REGION Network 3: E-Stop / Call: 运行 模式 area 1 - Create 新的 OpMode
   // 介绍：设置和管理操作操作模式OPMode，有几个OPMode就需要调用几次，每次调用都需要对其与HMI的关系进行定义。
   // 一个OPMode至少需要一个HMI/pannei控制；
   // 一个HMI/Panel可以控制多个OPMode；
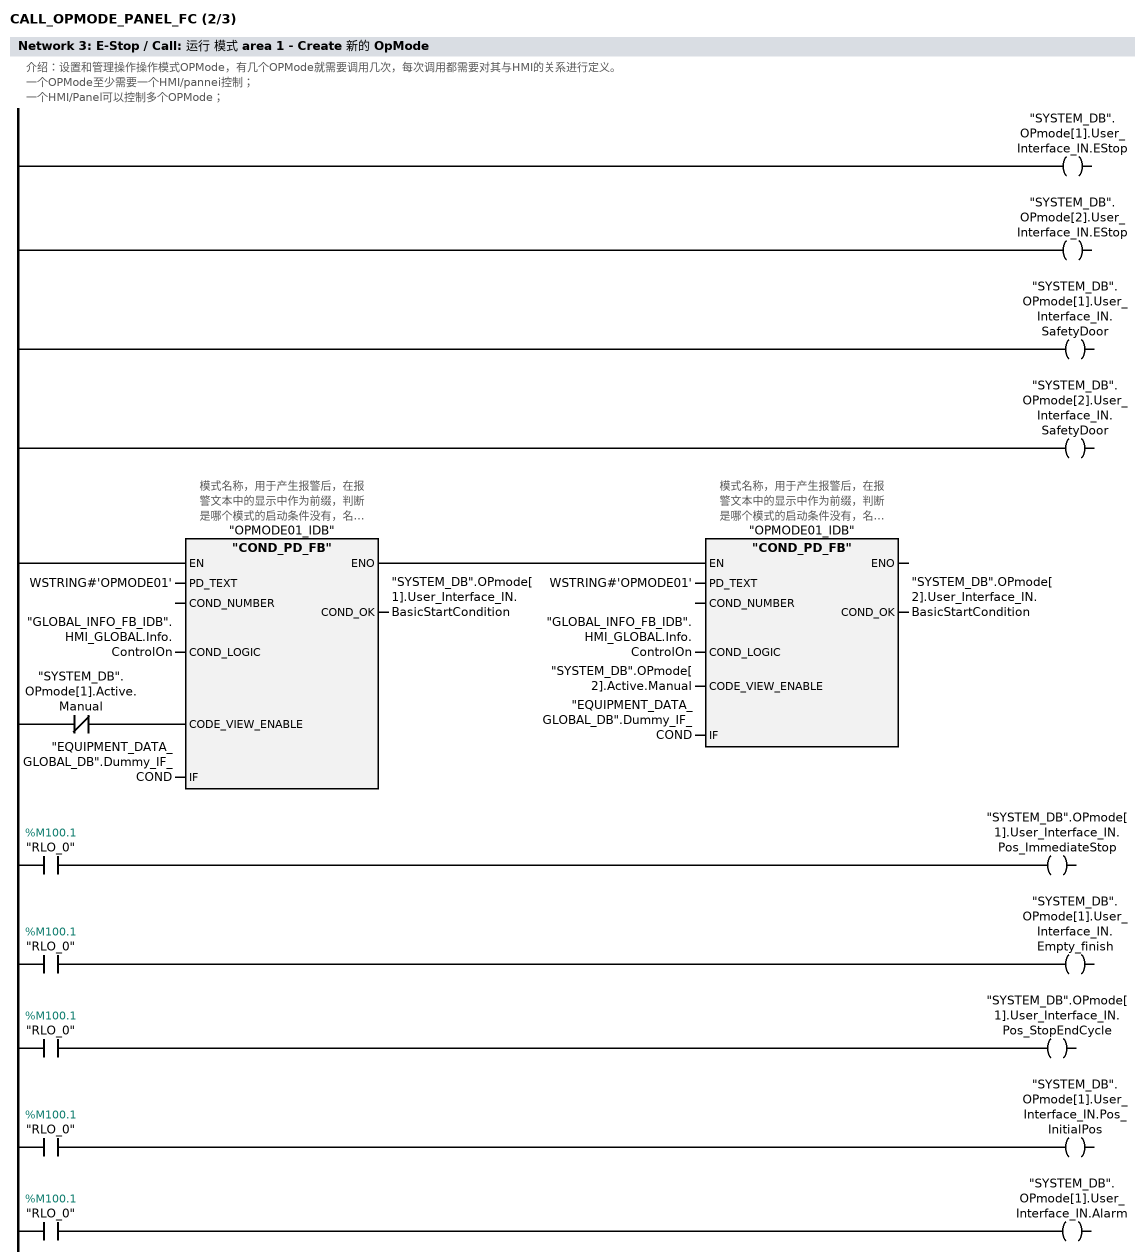
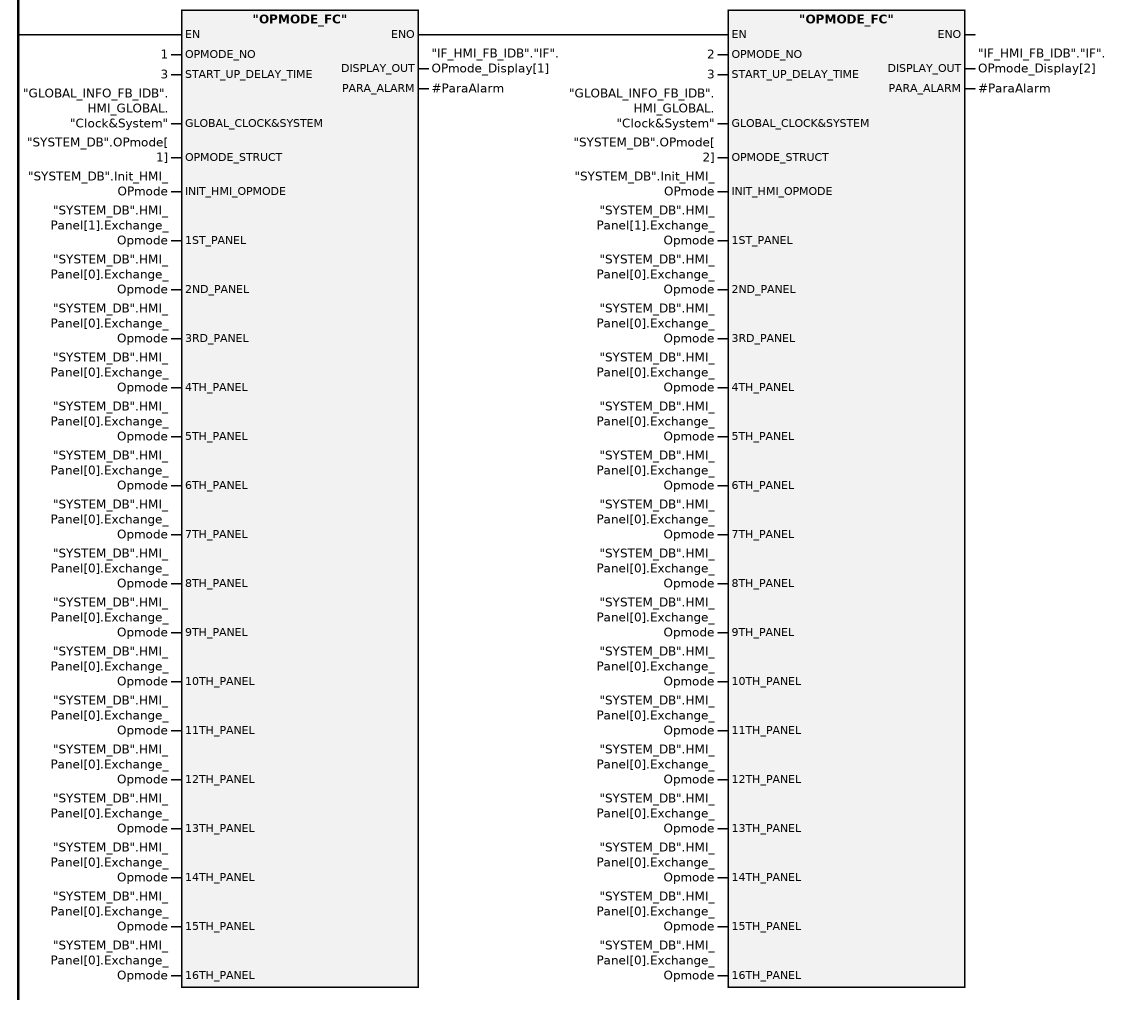
   RUNG wire#powerrail
      Coil( "SYSTEM_DB".OPmode[1].User_Interface_IN.EStop )
   END_RUNG
   RUNG wire#powerrail
      Coil( "SYSTEM_DB".OPmode[2].User_Interface_IN.EStop )
   END_RUNG
   RUNG wire#powerrail
      Coil( "SYSTEM_DB".OPmode[1].User_Interface_IN.SafetyDoor )
   END_RUNG
   RUNG wire#powerrail
      Coil( "SYSTEM_DB".OPmode[2].User_Interface_IN.SafetyDoor )
   END_RUNG
   RUNG wire#powerrail
      "OPMODE01_IDB"(CODE_VIEW_ENABLE := wire#w1, PD_TEXT := WSTRING#'OPMODE01', COND_NUMBER :=, COND_LOGIC := "GLOBAL_INFO_FB_IDB".HMI_GLOBAL.Info.ControlOn, "IF" := "EQUIPMENT_DATA_GLOBAL_DB".Dummy_IF_COND, COND_OK => "SYSTEM_DB".OPmode[1].User_Interface_IN.BasicStartCondition)   // 模式名称，用于产生报警后，在报警文本中的显示中作为前缀，判断是哪个模式的启动条件没有，名称已经预先填写在了对应DB块数据中
      "OPMODE01_IDB"(PD_TEXT := WSTRING#'OPMODE01', COND_NUMBER :=, COND_LOGIC := "GLOBAL_INFO_FB_IDB".HMI_GLOBAL.Info.ControlOn, CODE_VIEW_ENABLE := "SYSTEM_DB".OPmode[2].Active.Manual, "IF" := "EQUIPMENT_DATA_GLOBAL_DB".Dummy_IF_COND, COND_OK => "SYSTEM_DB".OPmode[2].User_Interface_IN.BasicStartCondition)   // 模式名称，用于产生报警后，在报警文本中的显示中作为前缀，判断是哪个模式的启动条件没有，名称已经预先填写在了对应DB块数据中
   END_RUNG
   RUNG wire#powerrail
      I_Contact( "SYSTEM_DB".OPmode[1].Active.Manual )
   END_RUNG wire#w1
   RUNG wire#powerrail
      Contact( "RLO_0" )
      Coil( "SYSTEM_DB".OPmode[1].User_Interface_IN.Pos_ImmediateStop )
   END_RUNG
   RUNG wire#powerrail
      Contact( "RLO_0" )
      Coil( "SYSTEM_DB".OPmode[1].User_Interface_IN.Empty_finish )
   END_RUNG
   RUNG wire#powerrail
      Contact( "RLO_0" )
      Coil( "SYSTEM_DB".OPmode[1].User_Interface_IN.Pos_StopEndCycle )
   END_RUNG
   RUNG wire#powerrail
      Contact( "RLO_0" )
      Coil( "SYSTEM_DB".OPmode[1].User_Interface_IN.Pos_InitialPos )
   END_RUNG
   RUNG wire#powerrail
      Contact( "RLO_0" )
      Coil( "SYSTEM_DB".OPmode[1].User_Interface_IN.Alarm )
   END_RUNG
   RUNG wire#powerrail
      "OPMODE_FC"(OPMODE_NO := 1, START_UP_DELAY_TIME := 3, "GLOBAL_CLOCK&SYSTEM" := "GLOBAL_INFO_FB_IDB".HMI_GLOBAL."Clock&System", OPMODE_STRUCT := "SYSTEM_DB".OPmode[1], INIT_HMI_OPMODE := "SYSTEM_DB".Init_HMI_OPmode, "1ST_PANEL" := "SYSTEM_DB".HMI_Panel[1].Exchange_Opmode, "2ND_PANEL" := "SYSTEM_DB".HMI_Panel[0].Exchange_Opmode, "3RD_PANEL" := "SYSTEM_DB".HMI_Panel[0].Exchange_Opmode, "4TH_PANEL" := "SYSTEM_DB".HMI_Panel[0].Exchange_Opmode, "5TH_PANEL" := "SYSTEM_DB".HMI_Panel[0].Exchange_Opmode, "6TH_PANEL" := "SYSTEM_DB".HMI_Panel[0].Exchange_Opmode, "7TH_PANEL" := "SYSTEM_DB".HMI_Panel[0].Exchange_Opmode, "8TH_PANEL" := "SYSTEM_DB".HMI_Panel[0].Exchange_Opmode, "9TH_PANEL" := "SYSTEM_DB".HMI_Panel[0].Exchange_Opmode, "10TH_PANEL" := "SYSTEM_DB".HMI_Panel[0].Exchange_Opmode, "11TH_PANEL" := "SYSTEM_DB".HMI_Panel[0].Exchange_Opmode, "12TH_PANEL" := "SYSTEM_DB".HMI_Panel[0].Exchange_Opmode, "13TH_PANEL" := "SYSTEM_DB".HMI_Panel[0].Exchange_Opmode, "14TH_PANEL" := "SYSTEM_DB".HMI_Panel[0].Exchange_Opmode, "15TH_PANEL" := "SYSTEM_DB".HMI_Panel[0].Exchange_Opmode, "16TH_PANEL" := "SYSTEM_DB".HMI_Panel[0].Exchange_Opmode, DISPLAY_OUT => "IF_HMI_FB_IDB"."IF".OPmode_Display[1], PARA_ALARM => #ParaAlarm)
      "OPMODE_FC"(OPMODE_NO := 2, START_UP_DELAY_TIME := 3, "GLOBAL_CLOCK&SYSTEM" := "GLOBAL_INFO_FB_IDB".HMI_GLOBAL."Clock&System", OPMODE_STRUCT := "SYSTEM_DB".OPmode[2], INIT_HMI_OPMODE := "SYSTEM_DB".Init_HMI_OPmode, "1ST_PANEL" := "SYSTEM_DB".HMI_Panel[1].Exchange_Opmode, "2ND_PANEL" := "SYSTEM_DB".HMI_Panel[0].Exchange_Opmode, "3RD_PANEL" := "SYSTEM_DB".HMI_Panel[0].Exchange_Opmode, "4TH_PANEL" := "SYSTEM_DB".HMI_Panel[0].Exchange_Opmode, "5TH_PANEL" := "SYSTEM_DB".HMI_Panel[0].Exchange_Opmode, "6TH_PANEL" := "SYSTEM_DB".HMI_Panel[0].Exchange_Opmode, "7TH_PANEL" := "SYSTEM_DB".HMI_Panel[0].Exchange_Opmode, "8TH_PANEL" := "SYSTEM_DB".HMI_Panel[0].Exchange_Opmode, "9TH_PANEL" := "SYSTEM_DB".HMI_Panel[0].Exchange_Opmode, "10TH_PANEL" := "SYSTEM_DB".HMI_Panel[0].Exchange_Opmode, "11TH_PANEL" := "SYSTEM_DB".HMI_Panel[0].Exchange_Opmode, "12TH_PANEL" := "SYSTEM_DB".HMI_Panel[0].Exchange_Opmode, "13TH_PANEL" := "SYSTEM_DB".HMI_Panel[0].Exchange_Opmode, "14TH_PANEL" := "SYSTEM_DB".HMI_Panel[0].Exchange_Opmode, "15TH_PANEL" := "SYSTEM_DB".HMI_Panel[0].Exchange_Opmode, "16TH_PANEL" := "SYSTEM_DB".HMI_Panel[0].Exchange_Opmode, DISPLAY_OUT => "IF_HMI_FB_IDB"."IF".OPmode_Display[2], PARA_ALARM => #ParaAlarm)
   END_RUNG
   // the same network as SCL:
   "SYSTEM_DB".OPmode[1].User_Interface_IN.EStop := TRUE;
   "SYSTEM_DB".OPmode[2].User_Interface_IN.EStop := TRUE;
   "SYSTEM_DB".OPmode[1].User_Interface_IN.SafetyDoor := TRUE;
   "SYSTEM_DB".OPmode[2].User_Interface_IN.SafetyDoor := TRUE;
   "OPMODE01_IDB"(PD_TEXT := WSTRING#'OPMODE01',   // "COND_PD_FB": 模式名称，用于产生报警后，在报警文本中的显示中作为前缀，判断是哪个模式的启动条件没有，名称已经预先填写在了对应DB块数据中
                  COND_LOGIC := "GLOBAL_INFO_FB_IDB".HMI_GLOBAL.Info.ControlOn,
                  CODE_VIEW_ENABLE := NOT "SYSTEM_DB".OPmode[1].Active.Manual,
                  "IF" := "EQUIPMENT_DATA_GLOBAL_DB".Dummy_IF_COND,
                  COND_OK => "SYSTEM_DB".OPmode[1].User_Interface_IN.BasicStartCondition,
                  ENO => #_w1);
   IF #_w1 THEN
       "OPMODE01_IDB"(PD_TEXT := WSTRING#'OPMODE01',   // "COND_PD_FB": 模式名称，用于产生报警后，在报警文本中的显示中作为前缀，判断是哪个模式的启动条件没有，名称已经预先填写在了对应DB块数据中
                      COND_LOGIC := "GLOBAL_INFO_FB_IDB".HMI_GLOBAL.Info.ControlOn,
                      CODE_VIEW_ENABLE := "SYSTEM_DB".OPmode[2].Active.Manual,
                      "IF" := "EQUIPMENT_DATA_GLOBAL_DB".Dummy_IF_COND,
                      COND_OK => "SYSTEM_DB".OPmode[2].User_Interface_IN.BasicStartCondition);
   END_IF;
   "SYSTEM_DB".OPmode[1].User_Interface_IN.Pos_ImmediateStop := "RLO_0";
   "SYSTEM_DB".OPmode[1].User_Interface_IN.Empty_finish := "RLO_0";
   "SYSTEM_DB".OPmode[1].User_Interface_IN.Pos_StopEndCycle := "RLO_0";
   "SYSTEM_DB".OPmode[1].User_Interface_IN.Pos_InitialPos := "RLO_0";
   "SYSTEM_DB".OPmode[1].User_Interface_IN.Alarm := "RLO_0";
   "OPMODE_FC"(OPMODE_NO := 1,
               START_UP_DELAY_TIME := 3,
               "GLOBAL_CLOCK&SYSTEM" := "GLOBAL_INFO_FB_IDB".HMI_GLOBAL."Clock&System",
               OPMODE_STRUCT := "SYSTEM_DB".OPmode[1],
               INIT_HMI_OPMODE := "SYSTEM_DB".Init_HMI_OPmode,
               "1ST_PANEL" := "SYSTEM_DB".HMI_Panel[1].Exchange_Opmode,
               "2ND_PANEL" := "SYSTEM_DB".HMI_Panel[0].Exchange_Opmode,
               "3RD_PANEL" := "SYSTEM_DB".HMI_Panel[0].Exchange_Opmode,
               "4TH_PANEL" := "SYSTEM_DB".HMI_Panel[0].Exchange_Opmode,
               "5TH_PANEL" := "SYSTEM_DB".HMI_Panel[0].Exchange_Opmode,
               "6TH_PANEL" := "SYSTEM_DB".HMI_Panel[0].Exchange_Opmode,
               "7TH_PANEL" := "SYSTEM_DB".HMI_Panel[0].Exchange_Opmode,
               "8TH_PANEL" := "SYSTEM_DB".HMI_Panel[0].Exchange_Opmode,
               "9TH_PANEL" := "SYSTEM_DB".HMI_Panel[0].Exchange_Opmode,
               "10TH_PANEL" := "SYSTEM_DB".HMI_Panel[0].Exchange_Opmode,
               "11TH_PANEL" := "SYSTEM_DB".HMI_Panel[0].Exchange_Opmode,
               "12TH_PANEL" := "SYSTEM_DB".HMI_Panel[0].Exchange_Opmode,
               "13TH_PANEL" := "SYSTEM_DB".HMI_Panel[0].Exchange_Opmode,
               "14TH_PANEL" := "SYSTEM_DB".HMI_Panel[0].Exchange_Opmode,
               "15TH_PANEL" := "SYSTEM_DB".HMI_Panel[0].Exchange_Opmode,
               "16TH_PANEL" := "SYSTEM_DB".HMI_Panel[0].Exchange_Opmode,
               DISPLAY_OUT => "IF_HMI_FB_IDB"."IF".OPmode_Display[1],
               PARA_ALARM => #ParaAlarm,
               ENO => #_w2);
   IF #_w2 THEN
       "OPMODE_FC"(OPMODE_NO := 2,
                   START_UP_DELAY_TIME := 3,
                   "GLOBAL_CLOCK&SYSTEM" := "GLOBAL_INFO_FB_IDB".HMI_GLOBAL."Clock&System",
                   OPMODE_STRUCT := "SYSTEM_DB".OPmode[2],
                   INIT_HMI_OPMODE := "SYSTEM_DB".Init_HMI_OPmode,
                   "1ST_PANEL" := "SYSTEM_DB".HMI_Panel[1].Exchange_Opmode,
                   "2ND_PANEL" := "SYSTEM_DB".HMI_Panel[0].Exchange_Opmode,
                   "3RD_PANEL" := "SYSTEM_DB".HMI_Panel[0].Exchange_Opmode,
                   "4TH_PANEL" := "SYSTEM_DB".HMI_Panel[0].Exchange_Opmode,
                   "5TH_PANEL" := "SYSTEM_DB".HMI_Panel[0].Exchange_Opmode,
                   "6TH_PANEL" := "SYSTEM_DB".HMI_Panel[0].Exchange_Opmode,
                   "7TH_PANEL" := "SYSTEM_DB".HMI_Panel[0].Exchange_Opmode,
                   "8TH_PANEL" := "SYSTEM_DB".HMI_Panel[0].Exchange_Opmode,
                   "9TH_PANEL" := "SYSTEM_DB".HMI_Panel[0].Exchange_Opmode,
                   "10TH_PANEL" := "SYSTEM_DB".HMI_Panel[0].Exchange_Opmode,
                   "11TH_PANEL" := "SYSTEM_DB".HMI_Panel[0].Exchange_Opmode,
                   "12TH_PANEL" := "SYSTEM_DB".HMI_Panel[0].Exchange_Opmode,
                   "13TH_PANEL" := "SYSTEM_DB".HMI_Panel[0].Exchange_Opmode,
                   "14TH_PANEL" := "SYSTEM_DB".HMI_Panel[0].Exchange_Opmode,
                   "15TH_PANEL" := "SYSTEM_DB".HMI_Panel[0].Exchange_Opmode,
                   "16TH_PANEL" := "SYSTEM_DB".HMI_Panel[0].Exchange_Opmode,
                   DISPLAY_OUT => "IF_HMI_FB_IDB"."IF".OPmode_Display[2],
                   PARA_ALARM => #ParaAlarm);
   END_IF;
END_REGION

REGION Network 4: Aufruf: HMI Schnittstelle / Call HMI_IF_FB
   // 介绍：HMI与PLC系统的接口功能块，
   // 此块用来管理所有的HMIheOPMode操作模式的接口，用户不需要对此做任何修改。
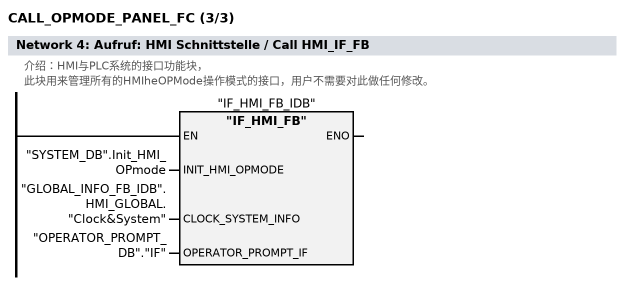
   RUNG wire#powerrail
      "IF_HMI_FB_IDB"(INIT_HMI_OPMODE := "SYSTEM_DB".Init_HMI_OPmode, CLOCK_SYSTEM_INFO := "GLOBAL_INFO_FB_IDB".HMI_GLOBAL."Clock&System", OPERATOR_PROMPT_IF := "OPERATOR_PROMPT_DB"."IF")
   END_RUNG
   // the same network as SCL:
   "IF_HMI_FB_IDB"(INIT_HMI_OPMODE := "SYSTEM_DB".Init_HMI_OPmode,   // "IF_HMI_FB"
                   CLOCK_SYSTEM_INFO := "GLOBAL_INFO_FB_IDB".HMI_GLOBAL."Clock&System",
                   OPERATOR_PROMPT_IF := "OPERATOR_PROMPT_DB"."IF");
END_REGION
END_FUNCTION

FUNCTION "IO映射" : Void   // FC4, LAD
{ S7_Optimized_Access := 'TRUE' }
// stored: SetENOAutomatically false
   VAR_TEMP
      LOOP : Int;
      Value : Byte;
      LOOP_1 : Int;
      Value_1 : Byte;
   END_VAR
BEGIN

REGION Network 1 (SCL)
   // 输入映射
   FOR #LOOP := 0 TO 10 BY 1 DO
       #Value := PEEK(area := 16#81, dbNumber := 0, byteOffset := #LOOP);
       POKE(area := 16#84,
            dbNumber := 12,
            byteOffset := #LOOP,
            value := #Value);
   END_FOR;
END_REGION

REGION Network 2 (SCL)
   // 输出映射
   FOR #LOOP_1 := 0 TO 8 BY 1 DO
       #Value_1 := PEEK(area := 16#84, dbNumber := 13, byteOffset := #LOOP_1);
       POKE(area := 16#82,
            dbNumber := 0,
            byteOffset := #LOOP_1,
            value := #Value_1);
   END_FOR;
END_REGION

REGION Network 3
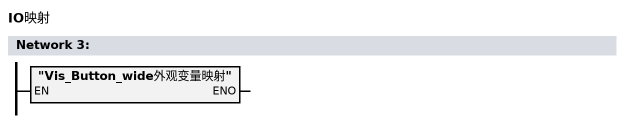
   RUNG wire#powerrail
      "Vis_Button_wide外观变量映射"()
   END_RUNG
   // the same network as SCL:
   "Vis_Button_wide外观变量映射"();
END_REGION
END_FUNCTION

FUNCTION "Vis_Button_wide外观变量映射" : Void   // FC5, LAD
{ S7_Optimized_Access := 'TRUE' }
// stored: SetENOAutomatically false
   VAR_TEMP
      x1 : Bool;
   END_VAR
BEGIN

REGION Network 1
   // 轴1轴2点动速度映射
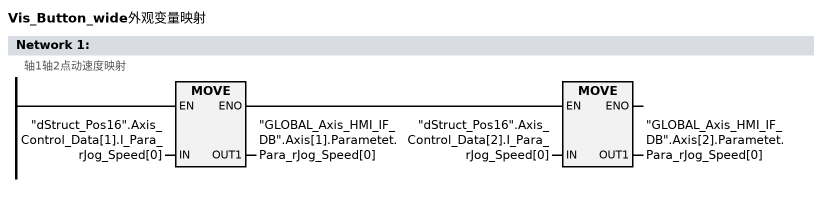
   RUNG wire#powerrail
      Move(in := "dStruct_Pos16".Axis_Control_Data[1].I_Para_rJog_Speed[0], out1 => "GLOBAL_Axis_HMI_IF_DB".Axis[1].Parametet.Para_rJog_Speed[0])
      Move(in := "dStruct_Pos16".Axis_Control_Data[2].I_Para_rJog_Speed[0], out1 => "GLOBAL_Axis_HMI_IF_DB".Axis[2].Parametet.Para_rJog_Speed[0])
   END_RUNG
   // the same network as SCL:
   "GLOBAL_Axis_HMI_IF_DB".Axis[1].Parametet.Para_rJog_Speed[0] := "dStruct_Pos16".Axis_Control_Data[1].I_Para_rJog_Speed[0];
   "GLOBAL_Axis_HMI_IF_DB".Axis[2].Parametet.Para_rJog_Speed[0] := "dStruct_Pos16".Axis_Control_Data[2].I_Para_rJog_Speed[0];
END_REGION

REGION Network 2 (SCL)
   "HMI变量汇总".Vis_Button_wideX1 := "IF_HMI_FB_IDB".IF.HMI[1].Vis_Button_wide.%X1;
   "HMI变量汇总".Vis_Button_wideX2 := "IF_HMI_FB_IDB".IF.HMI[1].Vis_Button_wide.%X2;
   "HMI变量汇总".Vis_Button_wideX3 := "IF_HMI_FB_IDB".IF.HMI[1].Vis_Button_wide.%X3;
   "HMI变量汇总".Vis_Button_wideX4 := "IF_HMI_FB_IDB".IF.HMI[1].Vis_Button_wide.%X4;
   "HMI变量汇总".Vis_Button_wideX5 := "IF_HMI_FB_IDB".IF.HMI[1].Vis_Button_wide.%X5;
   "HMI变量汇总".Vis_Button_wideX6 := "IF_HMI_FB_IDB".IF.HMI[1].Vis_Button_wide.%X6;
   "HMI变量汇总".Vis_Button_wideX7 := "IF_HMI_FB_IDB".IF.HMI[1].Vis_Button_wide.%X7;
   "HMI变量汇总".Vis_Button_wideX8 := "IF_HMI_FB_IDB".IF.HMI[1].Vis_Button_wide.%X8;
   "HMI变量汇总".Vis_Button_wideX9 := "IF_HMI_FB_IDB".IF.HMI[1].Vis_Button_wide.%X9;
   "HMI变量汇总".Vis_Button_wideX10 := "IF_HMI_FB_IDB".IF.HMI[1].Vis_Button_wide.%X10;
   "HMI变量汇总".Vis_Button_wideX11 := "IF_HMI_FB_IDB".IF.HMI[1].Vis_Button_wide.%X11;
   "HMI变量汇总".Vis_Button_wideX12 := "IF_HMI_FB_IDB".IF.HMI[1].Vis_Button_wide.%X12;

   "HMI变量汇总".Vis_Button_small1 := "IF_HMI_FB_IDB".IF.HMI[1].Vis_Button_small.%X1;
   "HMI变量汇总".Vis_Button_small2 := "IF_HMI_FB_IDB".IF.HMI[1].Vis_Button_small.%X2;
   "HMI变量汇总".Vis_Button_small3 := "IF_HMI_FB_IDB".IF.HMI[1].Vis_Button_small.%X3;
   "HMI变量汇总".Vis_Button_small4 := "IF_HMI_FB_IDB".IF.HMI[1].Vis_Button_small.%X4;
   "HMI变量汇总".Vis_Button_small5 := "IF_HMI_FB_IDB".IF.HMI[1].Vis_Button_small.%X5;
   "HMI变量汇总".Vis_Button_small6 := "IF_HMI_FB_IDB".IF.HMI[1].Vis_Button_small.%X6;
   "HMI变量汇总".Vis_Button_small7 := "IF_HMI_FB_IDB".IF.HMI[1].Vis_Button_small.%X7;
   "HMI变量汇总".Vis_Button_small8 := "IF_HMI_FB_IDB".IF.HMI[1].Vis_Button_small.%X8;
   "HMI变量汇总".Vis_Button_small9 := "IF_HMI_FB_IDB".IF.HMI[1].Vis_Button_small.%X9;
   "HMI变量汇总".Vis_Button_small10 := "IF_HMI_FB_IDB".IF.HMI[1].Vis_Button_small.%X10;
   "HMI变量汇总".Vis_Button_small11 := "IF_HMI_FB_IDB".IF.HMI[1].Vis_Button_small.%X11;
   "HMI变量汇总".Vis_Button_small12 := "IF_HMI_FB_IDB".IF.HMI[1].Vis_Button_small.%X12;




   #x1 := "IF_HMI_FB_IDB".IF.StateHeader_ForHMIAnimation[1].%X0;
   #x1 := "IF_HMI_FB_IDB".IF.StateHeader_ForHMIAnimation[1].%X1;
   #x1 := "IF_HMI_FB_IDB".IF.StateHeader_ForHMIAnimation[1].%X2;
   #x1 := "IF_HMI_FB_IDB".IF.StateHeader_ForHMIAnimation[1].%X3;
   #x1 := "IF_HMI_FB_IDB".IF.StateHeader_ForHMIAnimation[1].%X4;
   #x1 := "IF_HMI_FB_IDB".IF.StateHeader_ForHMIAnimation[1].%X5;
   #x1 := "IF_HMI_FB_IDB".IF.StateHeader_ForHMIAnimation[1].%X6;
   #x1 := "IF_HMI_FB_IDB".IF.StateHeader_ForHMIAnimation[1].%X7;
   #x1 := "IF_HMI_FB_IDB".IF.StateHeader_ForHMIAnimation[1].%X8;
   #x1 := "IF_HMI_FB_IDB".IF.StateHeader_ForHMIAnimation[1].%X9;
   #x1 := "IF_HMI_FB_IDB".IF.StateHeader_ForHMIAnimation[1].%X10;
   #x1 := "IF_HMI_FB_IDB".IF.StateHeader_ForHMIAnimation[1].%X11;
   #x1 := "IF_HMI_FB_IDB".IF.StateHeader_ForHMIAnimation[1].%X12;
   #x1 := "IF_HMI_FB_IDB".IF.StateHeader_ForHMIAnimation[1].%X13;
   #x1 := "IF_HMI_FB_IDB".IF.StateHeader_ForHMIAnimation[1].%X14;
   #x1 := "IF_HMI_FB_IDB".IF.StateHeader_ForHMIAnimation[1].%X15;
END_REGION
END_FUNCTION

FUNCTION "OPmode_01" : Void   // FC2, LAD
{ S7_Optimized_Access := 'TRUE' }
// stored: SetENOAutomatically false
BEGIN

REGION Network 1
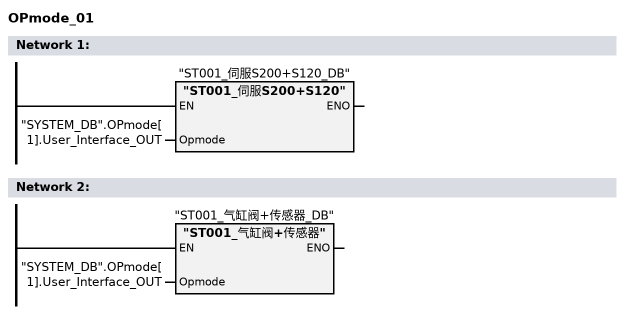
   RUNG wire#powerrail
      "ST001_伺服S200+S120_DB"(Opmode := "SYSTEM_DB".OPmode[1].User_Interface_OUT)
   END_RUNG
   // the same network as SCL:
   "ST001_伺服S200+S120_DB"(Opmode := "SYSTEM_DB".OPmode[1].User_Interface_OUT);   // "ST001_伺服S200+S120"
END_REGION

REGION Network 2
   RUNG wire#powerrail
      "ST001_气缸阀+传感器_DB"(Opmode := "SYSTEM_DB".OPmode[1].User_Interface_OUT)
   END_RUNG
   // the same network as SCL:
   "ST001_气缸阀+传感器_DB"(Opmode := "SYSTEM_DB".OPmode[1].User_Interface_OUT);   // "ST001_气缸阀+传感器"
END_REGION
END_FUNCTION

ORGANIZATION_BLOCK "CyclicInterrupt"   // OB30, LAD, CyclicInterrupt
{ S7_Optimized_Access := 'TRUE' }
// stored: SetENOAutomatically false
   VAR_INPUT
      Initial_Call : Bool;   // Initial call of this OB
      Event_Count : Int;   // Events discarded
   END_VAR
BEGIN

REGION Network 2
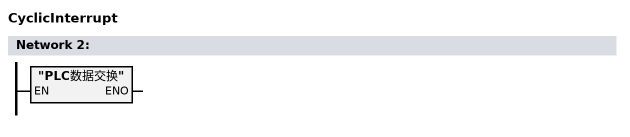
   RUNG wire#powerrail
      "PLC数据交换"()
   END_RUNG
   // the same network as SCL:
   "PLC数据交换"();
END_REGION
END_ORGANIZATION_BLOCK

FUNCTION "PLC数据交换" : Void   // FC1, LAD
{ S7_Optimized_Access := 'TRUE' }
// stored: SetENOAutomatically false
BEGIN

REGION Network 1
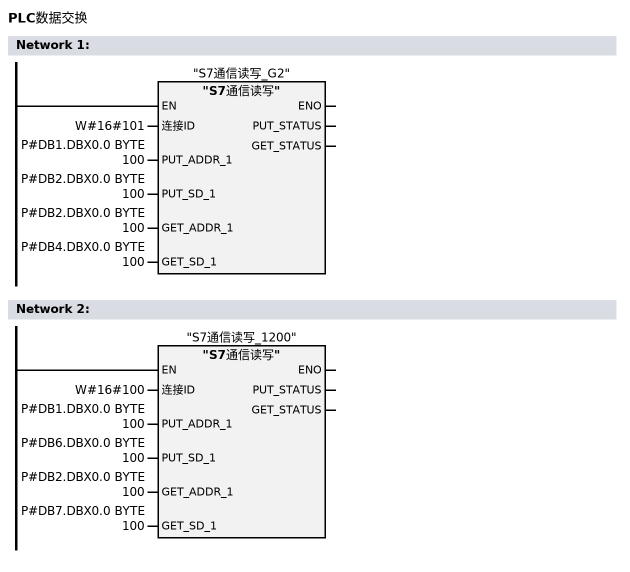
   RUNG wire#powerrail
      "S7通信读写_G2"(连接ID := W#16#101, PUT_ADDR_1 := P#DB1.DBX0.0 BYTE 100, PUT_SD_1 := P#DB2.DBX0.0 BYTE 100, GET_ADDR_1 := P#DB2.DBX0.0 BYTE 100, GET_SD_1 := P#DB4.DBX0.0 BYTE 100, PUT_STATUS =>, GET_STATUS =>)
   END_RUNG
   // the same network as SCL:
   "S7通信读写_G2"(连接ID := W#16#101,   // "S7通信读写"
               PUT_ADDR_1 := P#DB1.DBX0.0 BYTE 100,
               PUT_SD_1 := P#DB2.DBX0.0 BYTE 100,
               GET_ADDR_1 := P#DB2.DBX0.0 BYTE 100,
               GET_SD_1 := P#DB4.DBX0.0 BYTE 100);
END_REGION

REGION Network 2
   RUNG wire#powerrail
      "S7通信读写_1200"(连接ID := W#16#100, PUT_ADDR_1 := P#DB1.DBX0.0 BYTE 100, PUT_SD_1 := P#DB6.DBX0.0 BYTE 100, GET_ADDR_1 := P#DB2.DBX0.0 BYTE 100, GET_SD_1 := P#DB7.DBX0.0 BYTE 100, PUT_STATUS =>, GET_STATUS =>)
   END_RUNG
   // the same network as SCL:
   "S7通信读写_1200"(连接ID := W#16#100,   // "S7通信读写"
                 PUT_ADDR_1 := P#DB1.DBX0.0 BYTE 100,
                 PUT_SD_1 := P#DB6.DBX0.0 BYTE 100,
                 GET_ADDR_1 := P#DB2.DBX0.0 BYTE 100,
                 GET_SD_1 := P#DB7.DBX0.0 BYTE 100);
END_REGION
END_FUNCTION

FUNCTION_BLOCK "S7通信读写"   // FB1, LAD
{ S7_Optimized_Access := 'TRUE' }
// stored: MemoryReserve 100, SetENOAutomatically false
   VAR_INPUT
      连接ID : Word;
   END_VAR
   VAR_OUTPUT
      PUT_STATUS : Word;
      GET_STATUS : Word;
   END_VAR
   VAR_IN_OUT
      PUT_ADDR_1 : Remote;
      PUT_SD_1 : Variant;
      GET_ADDR_1 : Remote;
      GET_SD_1 : Variant;
   END_VAR
   VAR
      PUT_Instance { S7_SetPoint := 'True'} : PUT;
      GET_Instance { S7_SetPoint := 'True'} : GET;
      PUTdone : Bool;
      PUTerror : Bool;
      GETdone : Bool;
      GETerror : Bool;
   END_VAR
BEGIN

REGION Network 1
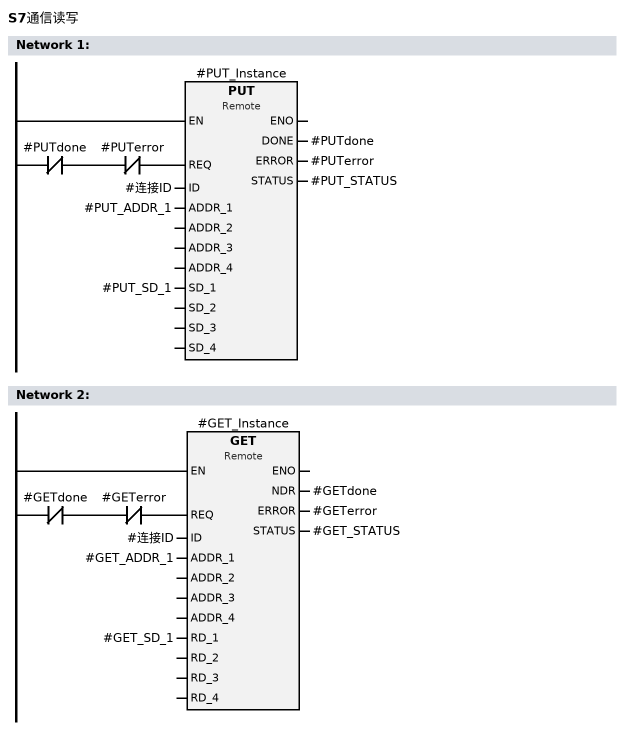
   RUNG wire#powerrail
      { S7_Templates := "[remote_type := Remote, local_type := Variant]" } #PUT_Instance.PUT(REQ := wire#w1, ID := #连接ID, ADDR_1 := #PUT_ADDR_1, ADDR_2 :=, ADDR_3 :=, ADDR_4 :=, SD_1 := #PUT_SD_1, SD_2 :=, SD_3 :=, SD_4 :=, DONE => #PUTdone, ERROR => #PUTerror, STATUS => #PUT_STATUS)
   END_RUNG
   RUNG wire#powerrail
      I_Contact( #PUTdone )
      I_Contact( #PUTerror )
   END_RUNG wire#w1
   // the same network as SCL:
   #PUT_Instance(REQ := NOT #PUTdone AND NOT #PUTerror,   // PUT
                 ID := #连接ID,
                 ADDR_1 := #PUT_ADDR_1,
                 SD_1 := #PUT_SD_1,
                 DONE => #PUTdone,
                 ERROR => #PUTerror,
                 STATUS => #PUT_STATUS);
END_REGION

REGION Network 2
   RUNG wire#powerrail
      { S7_Templates := "[remote_type := Remote, local_type := Variant]" } #GET_Instance.GET(REQ := wire#w1, ID := #连接ID, ADDR_1 := #GET_ADDR_1, ADDR_2 :=, ADDR_3 :=, ADDR_4 :=, RD_1 := #GET_SD_1, RD_2 :=, RD_3 :=, RD_4 :=, NDR => #GETdone, ERROR => #GETerror, STATUS => #GET_STATUS)
   END_RUNG
   RUNG wire#powerrail
      I_Contact( #GETdone )
      I_Contact( #GETerror )
   END_RUNG wire#w1
   // the same network as SCL:
   #GET_Instance(REQ := NOT #GETdone AND NOT #GETerror,   // GET
                 ID := #连接ID,
                 ADDR_1 := #GET_ADDR_1,
                 RD_1 := #GET_SD_1,
                 NDR => #GETdone,
                 ERROR => #GETerror,
                 STATUS => #GET_STATUS);
END_REGION
END_FUNCTION_BLOCK

FUNCTION "ST002示教台" : Void   // FC3, LAD
{ S7_Optimized_Access := 'TRUE' }
// stored: SetENOAutomatically false
BEGIN

REGION Network 1
   // IW256 G120状态字
   // IW258 G120当前频率（16#0-16#4000,对应0-50hz)
   // QW256 G120控制字
   // QW258 G120当前频率（16#0-16#4000,对应0-50hz)
END_REGION
END_FUNCTION

FUNCTION "FC_INPUT_MAP" : Void   // FC101, LAD
{ S7_Optimized_Access := 'TRUE' }
// stored: AutoNumber false, SetENOAutomatically false
   VAR_TEMP
      LOOP : Int;
      Value : Byte;
   END_VAR
BEGIN

REGION Network 1 (SCL): INPUT900BYTE
   FOR #LOOP := 0 TO 900 BY 1 DO
       #Value := PEEK(area := 16#81, dbNumber := 0, byteOffset := #LOOP);
       POKE(area:=16#84,dbNumber:=40, byteOffset:=#LOOP,value:=#Value);
   END_FOR;
END_REGION
END_FUNCTION

FUNCTION "FC_OUTPUT_MAP" : Void   // FC102, LAD
{ S7_Optimized_Access := 'TRUE' }
// stored: AutoNumber false, SetENOAutomatically false
   VAR_TEMP
      LOOP : Int;
      Value : Byte;
   END_VAR
BEGIN

REGION Network 1 (SCL): OUTPUT900BYTE
   FOR #LOOP := 0 TO 900 BY 1 DO
       #Value := PEEK(area := 16#84, dbNumber := 16, byteOffset := #LOOP);
       POKE(area:=16#82,dbNumber:=0, byteOffset:=#LOOP,value:=#Value);
   END_FOR;
END_REGION
END_FUNCTION

FUNCTION "DTLToString" : String   // FC20220, LAD
{ S7_Optimized_Access := 'TRUE' }
// stored: AutoNumber false, SetENOAutomatically false
   VAR_INPUT
      inDTL : DTL;   // Date as DTL tag
   END_VAR
   VAR_TEMP
      format : Bool;   // 1 = traditional, 0 = international
      separatorDate : Char;   // Separator between date components
      tempString : String;   // -
      tempSepTime : Char;   // -
      tempSepTimeNano : Char;   // -
      tempPosYear : USInt;   // -
      tempPosMonth : USInt;   // -
      tempPosDay : USInt;   // -
      tempPosHour : USInt;   // -
      tempPosMinute : USInt;   // -
      tempPosSecond : USInt;   // -
      tempPosNanosecond : USInt;   // -
      tempPosSepYearMonth : USInt;   // -
      tempPosSepMonthDay : USInt;   // -
      tempPosSepHourMinute : USInt;   // -
      tempPosSepMinuteSecond : USInt;   // -
      tempPosSepSecondNanosecond : USInt;   // -
      tempCount : Int;   // -
   END_VAR
BEGIN

REGION Network 1 (SCL): Initialization
   #tempString := '';
   #tempSepTime := ':';
   #tempSepTimeNano := '.';
   #format := 1;
END_REGION

REGION Network 2 (SCL): Set format parameters for output string
   IF  #format
   THEN                                          // International ISO 8601
       #tempPosYear := 1;                          // DTL  | Y| Y| Y| Y| -| M| M| -| D| D|  | H| H| :| M| M| :| S| S| .|NS|NS|NS|NS|NS|NS|NS|NS|NS
       #tempPosMonth := 6;                         // -----|--|--|--|--|--|--|--|--|--|--|--|--|--|--|--|--|--|--|--|--|--|--|--|--|--|--|--|--|--
       #tempPosDay := 9;                           // Pos  | 1| 2| 3| 4| 5| 6| 7| 8| 9|10|11|12|13|14|15|16|17|18|19|20|21|22|23|24|25|26|27|28|29
       #tempPosHour := 12;
       #tempPosMinute := 15;
       #tempPosSecond := 18;
       #tempPosNanosecond := 21;
       #tempPosSepYearMonth := 5;
       #tempPosSepMonthDay := 8;
       #tempPosSepHourMinute := 14;
       #tempPosSepMinuteSecond := 17;
       #tempPosSepSecondNanosecond := 20;
   ELSE                                          // Traditional (EU)
       #tempPosYear := 7;                          // DTL  | D| D| -| M| M| -| Y| Y| Y| Y|  | H| H| :| M| M| :| S| S| .|NS|NS|NS|NS|NS|NS|NS|NS|NS
       #tempPosMonth := 4;                         // -----|--|--|--|--|--|--|--|--|--|--|--|--|--|--|--|--|--|--|--|--|--|--|--|--|--|--|--|--|--
       #tempPosDay := 1;                           // Pos  | 1| 2| 3| 4| 5| 6| 7| 8| 9|10|11|12|13|14|15|16|17|18|19|20|21|22|23|24|25|26|27|28|29
       #tempPosHour := 12;
       #tempPosMinute := 15;
       #tempPosSecond := 18;
       #tempPosNanosecond := 21;
       #tempPosSepYearMonth := 6;
       #tempPosSepMonthDay := 3;
       #tempPosSepHourMinute := 14;
       #tempPosSepMinuteSecond := 17;
       #tempPosSepSecondNanosecond := 20;
   END_IF;
END_REGION

REGION Network 3 (SCL): Convert "Value" into "String" and place at the right position
   //==> DTL YEAR --> String --> #tempPosYear
   VAL_STRG(FORMAT := W#16#0000,
            IN := #inDTL.YEAR,
            P := #tempPosYear,
            PREC := 0,
            SIZE := 4,
            OUT => #tempString);    
   //==> DTL MONTH --> String --> #tempPosMonth
   VAL_STRG(FORMAT := W#16#0000,
            IN := #inDTL.MONTH,
            P := #tempPosMonth,
            PREC := 0,
            SIZE := 2,
            OUT => #tempString);     
   //==> DTL DAY --> String --> #tempPosDay
   VAL_STRG(FORMAT := W#16#0000,
            IN := #inDTL.DAY,
            P := #tempPosDay,
            PREC := 0,
            SIZE := 2,
            OUT => #tempString);    
   //==> DTL HOUR --> String --> #tempPosHour
   VAL_STRG(FORMAT := W#16#0000,
            IN := #inDTL.HOUR,
            P := #tempPosHour,
            PREC := 0,
            SIZE := 2,
            OUT => #tempString);     
   //==> DTL MINUTE --> String --> #tempPosMinute
   VAL_STRG(FORMAT := W#16#0000,
            IN := #inDTL.MINUTE,
            P := #tempPosMinute,
            PREC := 0,
            SIZE := 2,
            OUT => #tempString);     
   //==> DTL SECOND --> String --> #tempPosSecond
   VAL_STRG(FORMAT := W#16#0000,
            IN := #inDTL.SECOND,
            P := #tempPosSecond,
            PREC := 0,
            SIZE := 2,
            OUT => #tempString);     
   //==> // DTL NANOSECOND --> String --> #tempPosNanosecond
   VAL_STRG(FORMAT := W#16#0000,
            IN := #inDTL.NANOSECOND,
            P := #tempPosNanosecond,
            PREC := 0,
            SIZE := 9,
            OUT => #tempString);
END_REGION

REGION Network 4 (SCL): Place separators at the right position in the string
   #tempString[#tempPosSepYearMonth] := #separatorDate;
   #tempString[#tempPosSepMonthDay] := #separatorDate;
   #tempString[#tempPosSepHourMinute] := #tempSepTime;
   #tempString[#tempPosSepMinuteSecond] := #tempSepTime;
   #tempString[#tempPosSepSecondNanosecond] := #tempSepTimeNano;
END_REGION

REGION Network 5 (SCL): Correcting the string, due to the conversion of a leading "0" value into a "blank".-
   //==> Replacing of "blank" by "0"
   IF (#tempString[#tempPosMonth] = ' ')
   THEN
       #tempString[#tempPosMonth] := '0';
   END_IF;

   IF (#tempString[#tempPosDay] = ' ')
   THEN
       #tempString[#tempPosDay] := '0';
   END_IF;

   IF (#tempString[#tempPosHour] = ' ')
   THEN
       #tempString[#tempPosHour] := '0';
   END_IF;

   IF (#tempString[#tempPosMinute] = ' ')
   THEN
       #tempString[#tempPosMinute] := '0';
   END_IF;

   IF (#tempString[#tempPosSecond] = ' ')
   THEN
       #tempString[#tempPosSecond] := '0';
   END_IF;
END_REGION

REGION Network 6 (SCL): Temp count
   FOR #tempCount := 0 TO 5 BY 1
   DO
       IF (#tempString[#tempPosNanosecond + #tempCount] = ' ')
       THEN
           #tempString[#tempPosNanosecond + #tempCount] := '0';
       ELSE
           EXIT;
       END_IF;
   END_FOR;
END_REGION

REGION Network 7 (SCL): DTL to string
   #DTLToString := #tempString;
END_REGION
END_FUNCTION

FUNCTION "GenerateTransactionID" : Void   // FC20221, LAD
{ S7_Optimized_Access := 'TRUE' }
// stored: AutoNumber false, SetENOAutomatically false
   VAR_INPUT
      i_Start : Int;
   END_VAR
   VAR_OUTPUT
      dw_TransactionID : DWord;
   END_VAR
   VAR_TEMP
      i_Dummy : Int;
      t_DTL : DTL;
      i_CurrentYear : UInt;
      i_CurrentMonth : USInt;
      i_CurrentDay : USInt;
      i_CurrentHour : USInt;
      i_CurrentMinute : USInt;
      i_CurrentSecond : USInt;
      i_CurrentMilliSecond : UDInt;
      dw_CurrentYearToSecond : DWord;
      dw_CurrentMonthToSecond : DWord;
      dw_CurrentDayToSecond : DWord;
      dw_CurrentHourToSecond : DWord;
      dw_CurrentMinuteToSecond : DWord;
   END_VAR
BEGIN

REGION Network 1: Read time of day
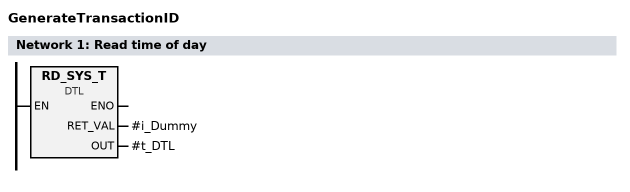
   RUNG wire#powerrail
      { S7_Templates := "date_type := DTL" } RD_SYS_T(RET_VAL => #i_Dummy, OUT => #t_DTL)
   END_RUNG
   // the same network as SCL:
   #i_Dummy := RD_SYS_T(OUT => #t_DTL);
END_REGION

REGION Network 2 (SCL): Generate unique values
   IF #i_Start = 1 THEN
       #i_CurrentYear := #t_DTL.YEAR;
       IF #i_CurrentYear > 1970 THEN
           #i_CurrentYear := #i_CurrentYear - 1970
           ;
       END_IF;//NEW

       #i_CurrentMonth := #t_DTL.MONTH;
       #i_CurrentDay := #t_DTL.DAY;
       #i_CurrentHour := #t_DTL.HOUR;
       #i_CurrentMinute := #t_DTL.MINUTE;
       #i_CurrentSecond := #t_DTL.SECOND;
       #i_CurrentMilliSecond := #t_DTL.NANOSECOND;

       #dw_CurrentYearToSecond := #i_CurrentYear * 31536000;
       #dw_CurrentMonthToSecond := #i_CurrentMonth * 2635200;
       #dw_CurrentDayToSecond := #i_CurrentDay * 86400;
       #dw_CurrentHourToSecond := #i_CurrentHour * 3600;
       #dw_CurrentMinuteToSecond := #i_CurrentMinute * 60;

       #dw_TransactionID := #dw_CurrentYearToSecond;
       #dw_TransactionID := #dw_TransactionID + #dw_CurrentMonthToSecond;
       #dw_TransactionID := #dw_TransactionID + #dw_CurrentDayToSecond;
       #dw_TransactionID := #dw_TransactionID + #dw_CurrentHourToSecond;
       #dw_TransactionID := #dw_TransactionID + #dw_CurrentMinuteToSecond;
       #dw_TransactionID := #dw_TransactionID + #i_CurrentSecond;
       #dw_TransactionID := #dw_TransactionID - #i_CurrentMilliSecond;

       IF #dw_TransactionID > 1620000000 THEN
           #dw_TransactionID := #dw_TransactionID - 1600000000;
       END_IF;

   ELSE
       #dw_TransactionID := 0;

   END_IF;
END_REGION
END_FUNCTION

FUNCTION "GetTransaction_ID" : Void   // FC20222, LAD
{ S7_Optimized_Access := 'TRUE' }
// stored: AutoNumber false, SetENOAutomatically false
   VAR_INPUT
      i_Start : Int;
   END_VAR
   VAR_OUTPUT
      oTransactionID : DWord;
   END_VAR
   VAR_TEMP
      i_Dummy : Int;
      t_DTL : DTL;
      tDTL_String : String;
      tDTL_LInt : LInt;
   END_VAR
   VAR_TEMP   // added for the SCL form of the ladder/FBD networks
      _w1 : Bool;
      _w2 : Bool;
      _w3 : Bool;
      _w4 : Bool;
      _w5 : Bool;
      _w6 : Bool;
   END_VAR
BEGIN

REGION Network 1: Read time of day
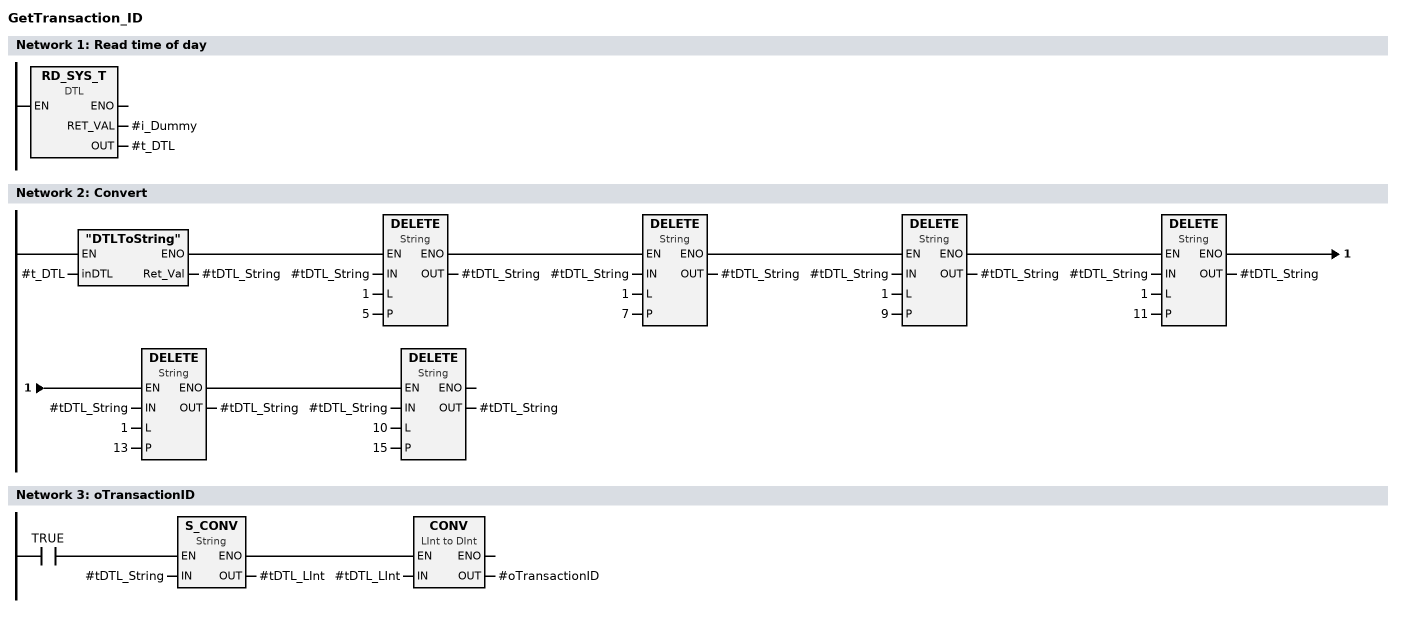
   RUNG wire#powerrail
      { S7_Templates := "date_type := DTL" } RD_SYS_T(RET_VAL => #i_Dummy, OUT => #t_DTL)
   END_RUNG
   // the same network as SCL:
   #i_Dummy := RD_SYS_T(OUT => #t_DTL);
END_REGION

REGION Network 2: Convert
   RUNG wire#powerrail
      "DTLToString"(inDTL := #t_DTL, Ret_Val => #tDTL_String)
      { S7_Templates := "str_type := String" } DELETE(IN := #tDTL_String, L := 1, P := 5, OUT => #tDTL_String)
      { S7_Templates := "str_type := String" } DELETE(IN := #tDTL_String, L := 1, P := 7, OUT => #tDTL_String)
      { S7_Templates := "str_type := String" } DELETE(IN := #tDTL_String, L := 1, P := 9, OUT => #tDTL_String)
      { S7_Templates := "str_type := String" } DELETE(IN := #tDTL_String, L := 1, P := 11, OUT => #tDTL_String)
      { S7_Templates := "str_type := String" } DELETE(IN := #tDTL_String, L := 1, P := 13, OUT => #tDTL_String)
      { S7_Templates := "str_type := String" } DELETE(IN := #tDTL_String, L := 10, P := 15, OUT => #tDTL_String)
   END_RUNG
   // the same network as SCL:
   #tDTL_String := "DTLToString"(inDTL := #t_DTL, ENO => #_w1);
   DELETE(EN := #_w1, IN := #tDTL_String, L := 1, P := 5, OUT => #tDTL_String, ENO => #_w2);
   DELETE(EN := #_w2, IN := #tDTL_String, L := 1, P := 7, OUT => #tDTL_String, ENO => #_w3);
   DELETE(EN := #_w3, IN := #tDTL_String, L := 1, P := 9, OUT => #tDTL_String, ENO => #_w4);
   DELETE(EN := #_w4, IN := #tDTL_String, L := 1, P := 11, OUT => #tDTL_String, ENO => #_w5);
   DELETE(EN := #_w5, IN := #tDTL_String, L := 1, P := 13, OUT => #tDTL_String, ENO => #_w6);
   IF #_w6 THEN DELETE(IN := #tDTL_String, L := 10, P := 15, OUT => #tDTL_String); END_IF;
END_REGION

REGION Network 3: oTransactionID
   RUNG wire#powerrail
      Contact( TRUE )
      { S7_Templates := "[src_type := String, dest_type := LInt]" } S_CONV(IN := #tDTL_String, OUT => #tDTL_LInt)
      { S7_Templates := "[SrcType := LInt, DestType := DInt]" } Convert(in := #tDTL_LInt, out => #oTransactionID)
   END_RUNG
   // the same network as SCL:
   S_CONV(EN := TRUE, IN := #tDTL_String, OUT => #tDTL_LInt, ENO => #_w1);
   IF #_w1 THEN #oTransactionID := LINT_TO_DINT(#tDTL_LInt); END_IF;
END_REGION
END_FUNCTION

FUNCTION "Start&EndTime" : Void   // FC20224, LAD
{ S7_Optimized_Access := 'FALSE' }
// stored: AutoNumber false, SetENOAutomatically false
   VAR_INPUT
      ReadEnable : Bool;
      SelectionIndex : Int;
      DB_Source : DB_ANY;
   END_VAR
   VAR_TEMP
      i_dummy : Int;
      i_DB_Source : Int;
      i_SourceSize : Int;
      i_StartAdressSource01 : Int;
      i_StartAdressSource02 : Int;
      di_AdressSource01 : DInt;
      di_AdressSource02 : DInt;
      pa_Any01 : Any;
      pa_Any02 : Any;
      t_DTL : DTL;
      StringOfTheCurrentTime : String[32];
   END_VAR
BEGIN

NETWORK
TITLE = Read time of day
      CALL  RD_SYS_T
      ( RET_VAL := #i_dummy,
        OUT     := #t_DTL
      );


NETWORK
TITLE = DTL to string
      CALL  "DTLToString"
      ( inDTL   := #t_DTL,
        Ret_Val := #StringOfTheCurrentTime
      );


NETWORK
TITLE = Init. Variables
      OPN   #DB_Source;
      L     DBNO;
      T     #i_DB_Source;

      L     838;
      T     #i_SourceSize;
//==> StartTime
      L     250;
      T     #i_StartAdressSource01;
//==> EndTime
      L     284;
      T     #i_StartAdressSource02;


NETWORK
TITLE = Write data
      A     #ReadEnable;
      JC    Y_VI;
      JU    N_VI;
Y_VI: NOP   0;
// STRUCTURE:
// BYTE 0  : 10h       -> S7
// BYTE 1  : 13h       -> String
// BYTE 2-3: Length of data
// BYTE 4-5: DB Number
// BYTE 6  : Area 84h=DB
// BYTE 6-8: Startadress

      L     #SelectionIndex;
      L     1;
      -D;
      L     #i_SourceSize;
      *D;
      L     #i_StartAdressSource01;
      +D;
      T     #di_AdressSource01;

      L     P##pa_Any01;
      LAR1;

      L     B#16#10;
      T     LB [AR1, P#0.0];
      L     B#16#2;
      T     LB [AR1, P#1.0];
      L     32;
      T     LW [AR1, P#2.0];
      L     #i_DB_Source;
      T     LW [AR1, P#4.0];
      L     #di_AdressSource01;
      SLD   3;
      OD    DW#16#84000000;
      T     LD [AR1, P#6.0];
//==>Copty to . . .
      CALL  BLKMOV
      ( SRCBLK  := #StringOfTheCurrentTime,
        RET_VAL := #i_dummy,
        DSTBLK  := #pa_Any01
      );


      L     #SelectionIndex;
      L     1;
      -D;
      L     #i_SourceSize;
      *D;
      L     #i_StartAdressSource02;
      +D;
      T     #di_AdressSource02;

      L     P##pa_Any02;
      LAR2;

      L     B#16#10;
      T     LB [AR2, P#0.0];
      L     B#16#2;
      T     LB [AR2, P#1.0];
      L     32;
      T     LW [AR2, P#2.0];
      L     #i_DB_Source;
      T     LW [AR2, P#4.0];
      L     #di_AdressSource02;
      SLD   3;
      OD    DW#16#84000000;
      T     LD [AR2, P#6.0];

//==>Copty to . . .
      CALL  BLKMOV
      ( SRCBLK  := #StringOfTheCurrentTime,
        RET_VAL := #i_dummy,
        DSTBLK  := #pa_Any02
      );

N_VI: NOP   0;
END_FUNCTION

FUNCTION "StringToDTL" : DTL   // FC20225, LAD
{ S7_Optimized_Access := 'TRUE' }
// stored: AutoNumber false, SetENOAutomatically false
   VAR_INPUT
      inString : String;   // Date as String tag
   END_VAR
   VAR_OUTPUT
      error : Bool;   // "0" = no error; "1" = error
      status : Word;   // status and error codes
   END_VAR
   VAR_TEMP
      format : Bool;   // Format of inString/ 0=traditional; 1=international
      tempCounter : Int;   // -
      tempOutput : DTL;   // -
      tempYear : String;   // -
      tempMonth : String;   // -
      tempDay : String;   // -
      tempHour : String;   // -
      tempMinute : String;   // -
      tempSecond : String;   // -
      tempNanosecond : String;   // -
      tempPosYear : USInt;   // -
      tempPosMonth : USInt;   // -
      tempPosDay : USInt;   // -
      tempPosHour : USInt;   // -
      tempPosMinute : USInt;   // -
      tempPosSecond : USInt;   // -
      tempPosNanosecond : USInt;   // -
      tempPosSepYearMonth : USInt;   // -
      tempPosSepMonthDay : USInt;   // -
      tempPosSepHourMinute : USInt;   // -
      tempPosSepMinuteSecond : USInt;   // -
      tempPosSepSecondNanosecond : USInt;   // -
   END_VAR
   VAR CONSTANT
      NO_ERROR : Word := 16#0000;   // -
      NO_CURRENT_JOBS : Word := 16#7000;   // -
      ERROR_FORMAT_YEAR : Word := 16#8201;   // -
      ERROR_FORMAT_MONTH : Word := 16#8202;   // -
      ERROR_FORMAT_DAY : Word := 16#8203;   // -
      ERROR_FORMAT_HOUR : Word := 16#8204;   // -
      ERROR_FORMAT_MINUTE : Word := 16#8205;   // -
      ERROR_FORMAT_SECOND : Word := 16#8206;   // -
      ERROR_FORMAT_NANOSECOND : Word := 16#8207;   // -
      INITIAL_VALUE : DTL := DTL#1970-01-01-00:00:00.0;   // -
   END_VAR
   // Ret_Val : Date as DTL tag
BEGIN

REGION Network 1 (SCL): Set initial parameters
   #error := FALSE;
   #status := #NO_ERROR;

   IF #inString = ''
   THEN
       #StringToDTL := #INITIAL_VALUE;
       #status := #NO_CURRENT_JOBS;
       RETURN;
   END_IF;

   #format := 1;
END_REGION

REGION Network 2 (SCL): Set format parameters for input string
   IF  #format
   THEN
       #tempPosYear := 1;                          // DTL  | Y| Y| Y| Y| -| M| M| -| D| D|  | H| H| :| M| M| :| S| S| .|NS|NS|NS|NS|NS|NS|NS|NS|NS
       #tempPosMonth := 6;                         // -----|--|--|--|--|--|--|--|--|--|--|--|--|--|--|--|--|--|--|--|--|--|--|--|--|--|--|--|--|--
       #tempPosDay := 9;                           // Pos  | 1| 2| 3| 4| 5| 6| 7| 8| 9|10|11|12|13|14|15|16|17|18|19|20|21|22|23|24|25|26|27|28|29
       #tempPosHour := 12;
       #tempPosMinute := 15;
       #tempPosSecond := 18;
       #tempPosNanosecond := 21;
       #tempPosSepYearMonth := 5;
       #tempPosSepMonthDay := 8;
       #tempPosSepHourMinute := 14;
       #tempPosSepMinuteSecond := 17;
       #tempPosSepSecondNanosecond := 20;
   ELSE
       #tempPosYear := 7;                          // DTL  | D| D| -| M| M| -| Y| Y| Y| Y|  | H| H| :| M| M| :| S| S| .|NS|NS|NS|NS|NS|NS|NS|NS|NS
       #tempPosMonth := 4;                         // -----|--|--|--|--|--|--|--|--|--|--|--|--|--|--|--|--|--|--|--|--|--|--|--|--|--|--|--|--|--
       #tempPosDay := 1;                           // Pos  | 1| 2| 3| 4| 5| 6| 7| 8| 9|10|11|12|13|14|15|16|17|18|19|20|21|22|23|24|25|26|27|28|29
       #tempPosHour := 12;
       #tempPosMinute := 15;
       #tempPosSecond := 18;
       #tempPosNanosecond := 21;
       #tempPosSepYearMonth := 6;
       #tempPosSepMonthDay := 3;
       #tempPosSepHourMinute := 14;
       #tempPosSepMinuteSecond := 17;
       #tempPosSepSecondNanosecond := 20;
   END_IF;
END_REGION

REGION Network 3 (SCL): Separating the input string into components of DTL
   #tempYear := MID(IN := #inString, L := 4, P := #tempPosYear);
   #tempMonth := MID(IN := #inString, L := 2, P := #tempPosMonth);
   #tempDay := MID(IN := #inString, L := 2, P := #tempPosDay);
   #tempHour := MID(IN := #inString, L := 2, P := #tempPosHour);
   #tempMinute := MID(IN := #inString, L := 2, P := #tempPosMinute);
   #tempSecond := MID(IN := #inString, L := 2, P := #tempPosSecond);
   #tempNanosecond := MID(IN := #inString, L := 9, P := #tempPosNanosecond);
END_REGION

REGION Network 4 (SCL): Replacing of the "blan" in the nanosecondstring by "0"
   //==> Effect:   xx.1 --> xx.1 AND NOT xx.1 --> xx.000000001
   FOR #tempCounter := 1 TO 9 BY 1
   DO
       IF #tempNanosecond[#tempCounter] = ' '
       THEN
           #tempNanosecond[#tempCounter] := '0';
       END_IF;
   END_FOR;
END_REGION

REGION Network 5 (SCL): Converting separated String components into DTL values
   STRG_VAL(FORMAT := W#16#0000,
            IN := #tempYear,
            OUT => #tempOutput.YEAR,
            P := 1);

   STRG_VAL(FORMAT := W#16#0000,
            IN := #tempMonth,
            OUT => #tempOutput.MONTH,
            P := 1);

   STRG_VAL(FORMAT := W#16#0000,
            IN := #tempDay,
            OUT => #tempOutput.DAY,
            P := 1);

   STRG_VAL(FORMAT := W#16#0000,
            IN := #tempHour,
            OUT => #tempOutput.HOUR,
            P := 1);

   STRG_VAL(FORMAT := W#16#0000,
            IN := #tempMinute,
            OUT => #tempOutput.MINUTE,
            P := 1);

   STRG_VAL(FORMAT := W#16#0000,
            IN := #tempSecond,
            OUT => #tempOutput.SECOND,
            P := 1);

   STRG_VAL(FORMAT := W#16#0000,
            IN := #tempNanosecond,
            OUT => #tempOutput.NANOSECOND,
            P := 1);
END_REGION

REGION Network 6 (SCL): Format check
   IF (#tempOutput.YEAR < 1970) OR (2262 < #tempOutput.YEAR)
   THEN
       #error := TRUE;
       #status := #ERROR_FORMAT_YEAR;
       #StringToDTL := #INITIAL_VALUE;
       RETURN;
   END_IF;

   IF (#tempOutput.MONTH < 1) OR (12 < #tempOutput.MONTH)
   THEN
       #error := TRUE;
       #status := #ERROR_FORMAT_MONTH;
       #StringToDTL := #INITIAL_VALUE;
       RETURN;
   END_IF;

   IF (#tempOutput.DAY < 1) OR (31 < #tempOutput.DAY)
   THEN
       #error := TRUE;
       #status := #ERROR_FORMAT_DAY;
       #StringToDTL := #INITIAL_VALUE;
       RETURN;
   END_IF;

   IF (#tempOutput.HOUR < 0) OR (23 < #tempOutput.HOUR)
   THEN
       #error := TRUE;
       #status := #ERROR_FORMAT_HOUR;
       #StringToDTL := #INITIAL_VALUE;
       RETURN;
   END_IF;

   IF (#tempOutput.MINUTE < 0) OR (59 < #tempOutput.MINUTE)
   THEN
       #error := TRUE;
       #status := #ERROR_FORMAT_MINUTE;
       #StringToDTL := #INITIAL_VALUE;
       RETURN;
   END_IF;

   IF (#tempOutput.SECOND < 0) OR (59 < #tempOutput.SECOND)
   THEN
       #error := TRUE;
       #status := #ERROR_FORMAT_SECOND;
       #StringToDTL := #INITIAL_VALUE;
       RETURN;
   END_IF;

   IF (#tempOutput.NANOSECOND < 0) OR (999999999 < #tempOutput.NANOSECOND)
   THEN
       #error := TRUE;
       #status := #ERROR_FORMAT_NANOSECOND;
       #StringToDTL := #INITIAL_VALUE;
       RETURN;
   END_IF;
END_REGION

REGION Network 7 (SCL): String to DTL
   #StringToDTL := #tempOutput;
END_REGION
END_FUNCTION

FUNCTION "Variable_ID" : Void   // FC20226, LAD
TITLE = Any pointer
{ S7_Optimized_Access := 'FALSE' }
// stored: AutoNumber false, SetENOAutomatically false
   VAR_INPUT
      ReadEnable : Bool;
      SelectionIndex : Int;
      VariableLength : Int;
      DB_Source : DB_ANY;
      SourceSize : Int;
      StartAdressSource : Int;
      DB_Destination : DB_ANY;
      DestinationSize : Int;
      StartAdressDestination : Int;
   END_VAR
   VAR_TEMP
      i_dummy : Int;
      i_DB_Source : Int;
      i_DB_Destination : Int;
      di_AdressSource : DInt;
      di_AdressDestination : DInt;
      pa_Any : Any;
      pa_OUT : Any;
   END_VAR
BEGIN

NETWORK
TITLE = Init. Variables
      L     0;
      T     #i_dummy;
//==>
      OPN   #DB_Source;
      L     DBNO;
      T     #i_DB_Source;

//==> OUT01
      OPN   #DB_Destination;
      L     DBNO;
      T     #i_DB_Destination;


NETWORK
TITLE = Read data
      A     #ReadEnable;
      JC    Y_VI;
      JU    N_VI;
Y_VI: NOP   0;
// STRUCTURE:
// BYTE 0  : 10h       -> S7
// BYTE 1  : 13h       -> String
// BYTE 2-3: Length of data
// BYTE 4-5: DB Number
// BYTE 6  : Area 84h=DB
// BYTE 6-8: Startadress

      L     #SelectionIndex;
      L     1;
      -D;
      L     #SourceSize;
      *D;
      L     #StartAdressSource;
      +D;
      T     #di_AdressSource;

      L     P##pa_Any;
      LAR1;

      L     B#16#10;
      T     LB [AR1, P#0.0];
      L     B#16#2;
      T     LB [AR1, P#1.0];
      L     #VariableLength;
      T     LW [AR1, P#2.0];
      L     #i_DB_Source;
      T     LW [AR1, P#4.0];
      L     #di_AdressSource;
      SLD   3;
      OD    DW#16#84000000;
      T     LD [AR1, P#6.0];
//==>
      L     #SelectionIndex;
      L     1;
      -D;
      L     #DestinationSize;
      *D;
      L     #StartAdressDestination;
      +D;
      T     #di_AdressDestination;

      L     P##pa_OUT;
      LAR2;

      L     B#16#10;
      T     LB [AR2, P#0.0];
      L     B#16#2;
      T     LB [AR2, P#1.0];
      L     #VariableLength;
      T     LW [AR2, P#2.0];
      L     #i_DB_Destination;
      T     LW [AR2, P#4.0];
      L     #di_AdressDestination;
      SLD   3;
      OD    DW#16#84000000;
      T     LD [AR2, P#6.0];

//==>Copty to . . .
      CALL  BLKMOV
      ( SRCBLK  := #pa_Any,
        RET_VAL := #i_dummy,
        DSTBLK  := #pa_OUT
      );

N_VI: NOP   0;
END_FUNCTION

FUNCTION_BLOCK "COMP_VAL_==_OR_FB"   // FB30380, LAD
TITLE = COMP_VAL_==_OR_FB
{ S7_Optimized_Access := 'TRUE' }
AUTHOR : SICAR
FAMILY : Miscellaneous
VERSION : 1.0
// Der Baustein vergleicht die Werte der Eingänge IN1...IN8 mit dem Wert des Eingangs COMPARE_VALUE und verodert diese Vergleiche. Ist mindestens einer der Werte von IN1...IN8 gleich mit COMPARE_VALUE, so wird der Wert von COMPARE_VALUE in den Output VALUE geschrieben. Andernfalls wird VALUE mit dem Wert 0 beschrieben.
// UseCase: Damit kann ein "Summensignal" gebildet werden, z.B. für Produktionsdaten "LimitValues", womit ein Button animiert werden kann (Button "ProdData", "Grenzwerte").
// The block compares the values of the inputs IN1 ... IN8 with the value of the input COMPARE_VALUE and OR-operation these comparisons. If at least one of the values of IN1 ... IN8 is equal with COMPARE_VALUE, the value of COMPARE_VALUE is written to output VALUE. Otherwise, VALUE is written with the value 0. 
// UseCase: With this, a "summary signal" can be formed, e.g. for production data "LimitValues", with which a button can be animated (Button "ProdData", "Limit Values").
// stored: AutoNumber false, MemoryReserve 100, SetENOAutomatically false
   VAR_INPUT
      COMPARE_VALUE { ExternalAccessible := 'False'; ExternalVisible := 'False'; ExternalWritable := 'False'} : DWord;
      IN1 { ExternalAccessible := 'False'; ExternalVisible := 'False'; ExternalWritable := 'False'} : DWord;
      IN2 { ExternalAccessible := 'False'; ExternalVisible := 'False'; ExternalWritable := 'False'} : DWord;
      IN3 { ExternalAccessible := 'False'; ExternalVisible := 'False'; ExternalWritable := 'False'} : DWord;
      IN4 { ExternalAccessible := 'False'; ExternalVisible := 'False'; ExternalWritable := 'False'} : DWord;
      IN5 { ExternalAccessible := 'False'; ExternalVisible := 'False'; ExternalWritable := 'False'} : DWord;
      IN6 { ExternalAccessible := 'False'; ExternalVisible := 'False'; ExternalWritable := 'False'} : DWord;
      IN7 { ExternalAccessible := 'False'; ExternalVisible := 'False'; ExternalWritable := 'False'} : DWord;
      IN8 { ExternalAccessible := 'False'; ExternalVisible := 'False'; ExternalWritable := 'False'} : DWord;
   END_VAR
   VAR_OUTPUT
      VALUE { ExternalAccessible := 'False'; ExternalVisible := 'False'; ExternalWritable := 'False'} : DWord;
   END_VAR
   VAR_TEMP
      Dummy : Bool;
   END_VAR
BEGIN

REGION Network 1: VALUE = 0 schreiben / set VALUE = 0
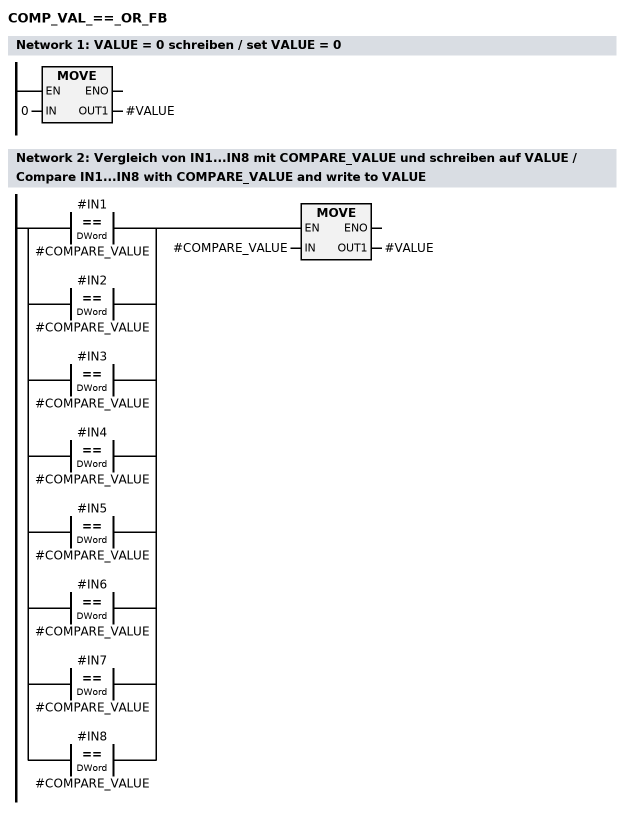
   RUNG wire#powerrail
      Move(in := 0, out1 => #VALUE)
   END_RUNG
   // the same network as SCL:
   #VALUE := 0;
END_REGION

REGION Network 2: Vergleich von IN1...IN8 mit COMPARE_VALUE und schreiben auf VALUE / Compare IN1...IN8 with COMPARE_VALUE and write to VALUE
   RUNG wire#powerrail
      { S7_Templates := "SrcType := DWord" } EQ_Contact(in1 := #IN1, in2 := #COMPARE_VALUE)
      wire#w1
      Move(in := #COMPARE_VALUE, out1 => #VALUE)
   END_RUNG
   RUNG wire#powerrail
      { S7_Templates := "SrcType := DWord" } EQ_Contact(in1 := #IN2, in2 := #COMPARE_VALUE)
   END_RUNG wire#w1
   RUNG wire#powerrail
      { S7_Templates := "SrcType := DWord" } EQ_Contact(in1 := #IN3, in2 := #COMPARE_VALUE)
   END_RUNG wire#w1
   RUNG wire#powerrail
      { S7_Templates := "SrcType := DWord" } EQ_Contact(in1 := #IN4, in2 := #COMPARE_VALUE)
   END_RUNG wire#w1
   RUNG wire#powerrail
      { S7_Templates := "SrcType := DWord" } EQ_Contact(in1 := #IN5, in2 := #COMPARE_VALUE)
   END_RUNG wire#w1
   RUNG wire#powerrail
      { S7_Templates := "SrcType := DWord" } EQ_Contact(in1 := #IN6, in2 := #COMPARE_VALUE)
   END_RUNG wire#w1
   RUNG wire#powerrail
      { S7_Templates := "SrcType := DWord" } EQ_Contact(in1 := #IN7, in2 := #COMPARE_VALUE)
   END_RUNG wire#w1
   RUNG wire#powerrail
      { S7_Templates := "SrcType := DWord" } EQ_Contact(in1 := #IN8, in2 := #COMPARE_VALUE)
   END_RUNG wire#w1
   // the same network as SCL:
   IF (#IN1 = #COMPARE_VALUE) OR (#IN2 = #COMPARE_VALUE) OR (#IN3 = #COMPARE_VALUE) OR (#IN4 = #COMPARE_VALUE) OR (#IN5 = #COMPARE_VALUE) OR (#IN6 = #COMPARE_VALUE) OR (#IN7 = #COMPARE_VALUE) OR (#IN8 = #COMPARE_VALUE) THEN
       #VALUE := #COMPARE_VALUE;
   END_IF;
END_REGION

NETWORK
TITLE = Baustein-Ende / End of block
// ENO immer "1" setzen mit SET & SAVE / ENO alwasy set "1" wtih SET & SAVE
      SET;
      SAVE;
END_FUNCTION_BLOCK

FUNCTION_BLOCK "FB2002_Axis_Function"   // FB2, LAD
{ S7_Optimized_Access := 'TRUE' }
// stored: MemoryReserve 100, SetENOAutomatically false
   VAR_INPUT
      Plant_Identifier { ExternalAccessible := 'False'; ExternalVisible := 'False'; ExternalWritable := 'False'} : WString[24];
      Opmode { ExternalAccessible := 'False'; ExternalVisible := 'False'; ExternalWritable := 'False'} : "OPMODE_OUT_UDT";
      TO_Pos_Axis : TO_PositioningAxis;
      Axis_Nr : Int;
      Axis_AbsNum : Int;
      I_SS_bHome : Bool;   // 原点传感器
      I_SS_bFW : Bool := TRUE;   // 前限位
      I_SS_bBW : Bool := TRUE;   // 后限位
      I_CMD_bEnableAxis : Bool;   // 使能
      I_CMD_bResetAxis : Bool;   // 复位
      I_CMD_bjogForward : Bool;   // Taster Aufwärts / 正点
      I_CMD_bjogBackward : Bool;   // Taster Abwärts / 反点
      I_CMD_bmoveVelocity : Bool;   // 速度运行
      I_CMD_bstop : Bool;   // 停止
      I_CMD_bfastStop : Bool;   // 急停
      I_CMD_bHoming : Bool;   // 回零
      I_CMD_bGoToPos : Array[0..15] of Bool;   // Start Aufwärts in Automatik / 16个定位
      I_CMD_iGoToPos : Word;   // 16个定位 Word
      I_CMD_bCallAbsPos : Bool;   // 定位位置切换时，单独的定位按钮
      I_CMD_bRelPos : Bool;   // 相对定位
      I_InLock_bEnableAxis : Bool;   // 使能
      I_InLock_bResetAxis : Bool;   // 复位
      I_InLock_bjogForward : Bool;   // Taster Aufwärts / 正点
      I_InLock_bjogBackward : Bool;   // Taster Abwärts / 反点
      I_InLock_bmoveVelocity : Bool;   // 速度运行
      I_InLock_bstop : Bool;   // 停止
      I_InLock_bfastStop : Bool;   // 急停
      I_InLock_bHoming : Bool;   // 回零
      I_InLock_bGoToPos : Array[0..16] of Bool;   // Start Aufwärts in Automatik / 16个定位
      I_InLock_iGoToPos : Word;   // 16个定位 Word
      I_InLock_bCallAbsPos : Bool;   // 定位位置切换时，单独的定位按钮
      I_InLock_bRelPos : Bool;   // 相对定位
      I_InLock_MyBool : Array[0..5] of Bool;   // 临时变量
      I_CMD_bGoToPos_0 : Bool;   // Start Aufwärts in Automatik / 16个定位自动
      I_InLock_bGoToPos_0 : Bool;   // Start Aufwärts in Automatik / 16个定位条件
      I_CMD_bGoToPos_1 : Bool;   // Start Aufwärts in Automatik / 16个定位自动
      I_InLock_bGoToPos_1 : Bool;   // Start Aufwärts in Automatik / 16个定位条件
      I_CMD_bGoToPos_2 : Bool;   // Start Aufwärts in Automatik / 16个定位自动
      I_InLock_bGoToPos_2 : Bool;   // Start Aufwärts in Automatik / 16个定位条件
      I_CMD_bGoToPos_3 : Bool;   // Start Aufwärts in Automatik / 16个定位自动
      I_InLock_bGoToPos_3 : Bool;   // Start Aufwärts in Automatik / 16个定位条件
      I_CMD_bGoToPos_4 : Bool;   // Start Aufwärts in Automatik / 16个定位自动
      I_InLock_bGoToPos_4 : Bool;   // Start Aufwärts in Automatik / 16个定位条件
      I_CMD_bGoToPos_5 : Bool;   // Start Aufwärts in Automatik / 16个定位自动
      I_InLock_bGoToPos_5 : Bool;   // Start Aufwärts in Automatik / 16个定位条件
      I_CMD_bGoToPos_6 : Bool;   // Start Aufwärts in Automatik / 16个定位自动
      I_InLock_bGoToPos_6 : Bool;   // Start Aufwärts in Automatik / 16个定位条件
      I_CMD_bGoToPos_7 : Bool;   // Start Aufwärts in Automatik / 16个定位自动
      I_InLock_bGoToPos_7 : Bool;   // Start Aufwärts in Automatik / 16个定位条件
      I_CMD_bGoToPos_8 : Bool;   // Start Aufwärts in Automatik / 16个定位自动
      I_InLock_bGoToPos_8 : Bool;   // Start Aufwärts in Automatik / 16个定位条件
   END_VAR
   VAR_OUTPUT
      O_Status_bAxisReady : Bool;   // 轴通讯正常
      O_Status_bAxisEnabled : Bool;   // 轴使能
      O_Status_bjogForward : Bool;   // 轴正点中
      O_Status_bjogBackward : Bool;   // 轴反点中
      O_Status_bHomed : Bool;   // 轴归零完成
      O_Status_bAtHome : Bool;   // 轴在零位
      O_Status_bSstill : Bool;   // 轴静止
      O_Status_bAxisBusy : Bool;   // 轴运行中
      O_Status_bAxisSyned : Bool;   // 同步上
      O_Status_bAxisError : Bool;   // 轴报警
      O_Status_bAtPos : Array[0..15] of Bool;   // Ausgang Aufwärts / 在目标位置上
      O_Status_bPosDone : Array[0..15] of Bool;   // 定位完成
      O_Status_bPosing : Array[0..15] of Bool;   // Ausgang Aufwärts / 定位中
      O_Status_bRelPosDone : Bool;   // 相对定位完成
      O_Status_rActPos : LReal;   // 实际位置
      O_Status_rActSpeed : LReal;   // 实际速度
      O_Status_iAxisFaultNum : UDInt;   // 轴报警代码
      O_Status_iDriveFaultNum : UDInt;   // 驱动报警代码
      O_Status_iFBStatus : Word;   // 运动功能块状态
      O_Status_iMCStatus : Word;   // 运动指令状态
      O_Status_rDriveTorque : LReal;   // 驱动扭矩
      O_Status_rDriveTemp : LReal;   // 驱动温度
      O_Status_rDriveRpm : LReal;   // 驱动转速
      O_Status_AxisName : WString[24] := WSTRING#'No axis';   // Name of axis
      O_Status_mybool : Array[0..5] of Bool;   // 备用
      O_Status_myLreal : Array[0..5] of LReal;   // 备用
   END_VAR
   VAR_IN_OUT
      IF_HMI : "Axis_IF_HMI";
   END_VAR
   VAR
      myFB_Pos16_Ax01 { S7_SetPoint := 'True'} : "FB_Pos16_IO";
      Axis_01 { S7_SetPoint := 'True'} : "FB_Axis";
      i { ExternalAccessible := 'False'; ExternalVisible := 'False'; ExternalWritable := 'False'} : Int;
      j { ExternalAccessible := 'False'; ExternalVisible := 'False'; ExternalWritable := 'False'} : Int;
      HOMIEDONE : Bool;
   END_VAR
BEGIN

REGION Network 1
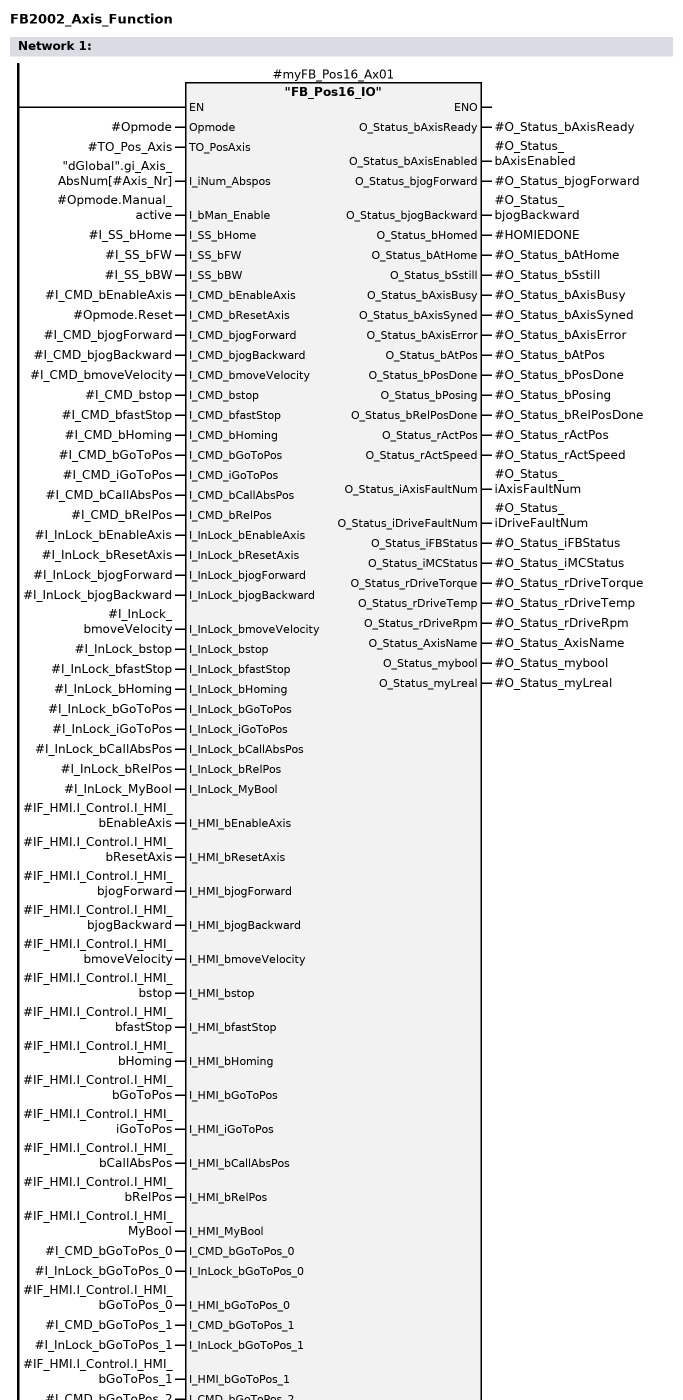
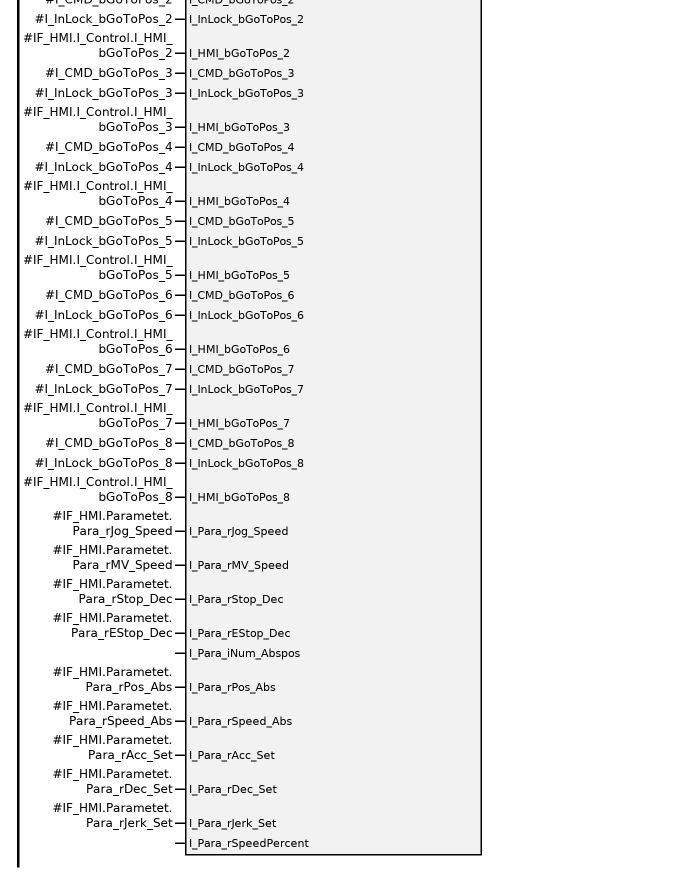
   RUNG wire#powerrail
      #myFB_Pos16_Ax01(Opmode := #Opmode, TO_PosAxis := #TO_Pos_Axis, I_iNum_Abspos := "dGlobal".gi_Axis_AbsNum[#Axis_Nr], I_bMan_Enable := #Opmode.Manual_active, I_SS_bHome := #I_SS_bHome, I_SS_bFW := #I_SS_bFW, I_SS_bBW := #I_SS_bBW, I_CMD_bEnableAxis := #I_CMD_bEnableAxis, I_CMD_bResetAxis := #Opmode.Reset, I_CMD_bjogForward := #I_CMD_bjogForward, I_CMD_bjogBackward := #I_CMD_bjogBackward, I_CMD_bmoveVelocity := #I_CMD_bmoveVelocity, I_CMD_bstop := #I_CMD_bstop, I_CMD_bfastStop := #I_CMD_bfastStop, I_CMD_bHoming := #I_CMD_bHoming, I_CMD_bGoToPos := #I_CMD_bGoToPos, I_CMD_iGoToPos := #I_CMD_iGoToPos, I_CMD_bCallAbsPos := #I_CMD_bCallAbsPos, I_CMD_bRelPos := #I_CMD_bRelPos, I_InLock_bEnableAxis := #I_InLock_bEnableAxis, I_InLock_bResetAxis := #I_InLock_bResetAxis, I_InLock_bjogForward := #I_InLock_bjogForward, I_InLock_bjogBackward := #I_InLock_bjogBackward, I_InLock_bmoveVelocity := #I_InLock_bmoveVelocity, I_InLock_bstop := #I_InLock_bstop, I_InLock_bfastStop := #I_InLock_bfastStop, I_InLock_bHoming := #I_InLock_bHoming, I_InLock_bGoToPos := #I_InLock_bGoToPos, I_InLock_iGoToPos := #I_InLock_iGoToPos, I_InLock_bCallAbsPos := #I_InLock_bCallAbsPos, I_InLock_bRelPos := #I_InLock_bRelPos, I_InLock_MyBool := #I_InLock_MyBool, I_HMI_bEnableAxis := #IF_HMI.I_Control.I_HMI_bEnableAxis, I_HMI_bResetAxis := #IF_HMI.I_Control.I_HMI_bResetAxis, I_HMI_bjogForward := #IF_HMI.I_Control.I_HMI_bjogForward, I_HMI_bjogBackward := #IF_HMI.I_Control.I_HMI_bjogBackward, I_HMI_bmoveVelocity := #IF_HMI.I_Control.I_HMI_bmoveVelocity, I_HMI_bstop := #IF_HMI.I_Control.I_HMI_bstop, I_HMI_bfastStop := #IF_HMI.I_Control.I_HMI_bfastStop, I_HMI_bHoming := #IF_HMI.I_Control.I_HMI_bHoming, I_HMI_bGoToPos := #IF_HMI.I_Control.I_HMI_bGoToPos, I_HMI_iGoToPos := #IF_HMI.I_Control.I_HMI_iGoToPos, I_HMI_bCallAbsPos := #IF_HMI.I_Control.I_HMI_bCallAbsPos, I_HMI_bRelPos := #IF_HMI.I_Control.I_HMI_bRelPos, I_HMI_MyBool := #IF_HMI.I_Control.I_HMI_MyBool, I_CMD_bGoToPos_0 := #I_CMD_bGoToPos_0, I_InLock_bGoToPos_0 := #I_InLock_bGoToPos_0, I_HMI_bGoToPos_0 := #IF_HMI.I_Control.I_HMI_bGoToPos_0, I_CMD_bGoToPos_1 := #I_CMD_bGoToPos_1, I_InLock_bGoToPos_1 := #I_InLock_bGoToPos_1, I_HMI_bGoToPos_1 := #IF_HMI.I_Control.I_HMI_bGoToPos_1, I_CMD_bGoToPos_2 := #I_CMD_bGoToPos_2, I_InLock_bGoToPos_2 := #I_InLock_bGoToPos_2, I_HMI_bGoToPos_2 := #IF_HMI.I_Control.I_HMI_bGoToPos_2, I_CMD_bGoToPos_3 := #I_CMD_bGoToPos_3, I_InLock_bGoToPos_3 := #I_InLock_bGoToPos_3, I_HMI_bGoToPos_3 := #IF_HMI.I_Control.I_HMI_bGoToPos_3, I_CMD_bGoToPos_4 := #I_CMD_bGoToPos_4, I_InLock_bGoToPos_4 := #I_InLock_bGoToPos_4, I_HMI_bGoToPos_4 := #IF_HMI.I_Control.I_HMI_bGoToPos_4, I_CMD_bGoToPos_5 := #I_CMD_bGoToPos_5, I_InLock_bGoToPos_5 := #I_InLock_bGoToPos_5, I_HMI_bGoToPos_5 := #IF_HMI.I_Control.I_HMI_bGoToPos_5, I_CMD_bGoToPos_6 := #I_CMD_bGoToPos_6, I_InLock_bGoToPos_6 := #I_InLock_bGoToPos_6, I_HMI_bGoToPos_6 := #IF_HMI.I_Control.I_HMI_bGoToPos_6, I_CMD_bGoToPos_7 := #I_CMD_bGoToPos_7, I_InLock_bGoToPos_7 := #I_InLock_bGoToPos_7, I_HMI_bGoToPos_7 := #IF_HMI.I_Control.I_HMI_bGoToPos_7, I_CMD_bGoToPos_8 := #I_CMD_bGoToPos_8, I_InLock_bGoToPos_8 := #I_InLock_bGoToPos_8, I_HMI_bGoToPos_8 := #IF_HMI.I_Control.I_HMI_bGoToPos_8, I_Para_rJog_Speed := #IF_HMI.Parametet.Para_rJog_Speed, I_Para_rMV_Speed := #IF_HMI.Parametet.Para_rMV_Speed, I_Para_rStop_Dec := #IF_HMI.Parametet.Para_rStop_Dec, I_Para_rEStop_Dec := #IF_HMI.Parametet.Para_rEStop_Dec, I_Para_iNum_Abspos :=, I_Para_rPos_Abs := #IF_HMI.Parametet.Para_rPos_Abs, I_Para_rSpeed_Abs := #IF_HMI.Parametet.Para_rSpeed_Abs, I_Para_rAcc_Set := #IF_HMI.Parametet.Para_rAcc_Set, I_Para_rDec_Set := #IF_HMI.Parametet.Para_rDec_Set, I_Para_rJerk_Set := #IF_HMI.Parametet.Para_rJerk_Set, I_Para_rSpeedPercent :=, O_Status_bAxisReady => #O_Status_bAxisReady, O_Status_bAxisEnabled => #O_Status_bAxisEnabled, O_Status_bjogForward => #O_Status_bjogForward, O_Status_bjogBackward => #O_Status_bjogBackward, O_Status_bHomed => #HOMIEDONE, O_Status_bAtHome => #O_Status_bAtHome, O_Status_bSstill => #O_Status_bSstill, O_Status_bAxisBusy => #O_Status_bAxisBusy, O_Status_bAxisSyned => #O_Status_bAxisSyned, O_Status_bAxisError => #O_Status_bAxisError, O_Status_bAtPos => #O_Status_bAtPos, O_Status_bPosDone => #O_Status_bPosDone, O_Status_bPosing => #O_Status_bPosing, O_Status_bRelPosDone => #O_Status_bRelPosDone, O_Status_rActPos => #O_Status_rActPos, O_Status_rActSpeed => #O_Status_rActSpeed, O_Status_iAxisFaultNum => #O_Status_iAxisFaultNum, O_Status_iDriveFaultNum => #O_Status_iDriveFaultNum, O_Status_iFBStatus => #O_Status_iFBStatus, O_Status_iMCStatus => #O_Status_iMCStatus, O_Status_rDriveTorque => #O_Status_rDriveTorque, O_Status_rDriveTemp => #O_Status_rDriveTemp, O_Status_rDriveRpm => #O_Status_rDriveRpm, O_Status_AxisName => #O_Status_AxisName, O_Status_mybool => #O_Status_mybool, O_Status_myLreal => #O_Status_myLreal)
   END_RUNG
   // the same network as SCL:
   #myFB_Pos16_Ax01(Opmode := #Opmode,   // "FB_Pos16_IO"
                    TO_PosAxis := #TO_Pos_Axis,
                    I_iNum_Abspos := "dGlobal".gi_Axis_AbsNum[#Axis_Nr],
                    I_bMan_Enable := #Opmode.Manual_active,
                    I_SS_bHome := #I_SS_bHome,
                    I_SS_bFW := #I_SS_bFW,
                    I_SS_bBW := #I_SS_bBW,
                    I_CMD_bEnableAxis := #I_CMD_bEnableAxis,
                    I_CMD_bResetAxis := #Opmode.Reset,
                    I_CMD_bjogForward := #I_CMD_bjogForward,
                    I_CMD_bjogBackward := #I_CMD_bjogBackward,
                    I_CMD_bmoveVelocity := #I_CMD_bmoveVelocity,
                    I_CMD_bstop := #I_CMD_bstop,
                    I_CMD_bfastStop := #I_CMD_bfastStop,
                    I_CMD_bHoming := #I_CMD_bHoming,
                    I_CMD_bGoToPos := #I_CMD_bGoToPos,
                    I_CMD_iGoToPos := #I_CMD_iGoToPos,
                    I_CMD_bCallAbsPos := #I_CMD_bCallAbsPos,
                    I_CMD_bRelPos := #I_CMD_bRelPos,
                    I_InLock_bEnableAxis := #I_InLock_bEnableAxis,
                    I_InLock_bResetAxis := #I_InLock_bResetAxis,
                    I_InLock_bjogForward := #I_InLock_bjogForward,
                    I_InLock_bjogBackward := #I_InLock_bjogBackward,
                    I_InLock_bmoveVelocity := #I_InLock_bmoveVelocity,
                    I_InLock_bstop := #I_InLock_bstop,
                    I_InLock_bfastStop := #I_InLock_bfastStop,
                    I_InLock_bHoming := #I_InLock_bHoming,
                    I_InLock_bGoToPos := #I_InLock_bGoToPos,
                    I_InLock_iGoToPos := #I_InLock_iGoToPos,
                    I_InLock_bCallAbsPos := #I_InLock_bCallAbsPos,
                    I_InLock_bRelPos := #I_InLock_bRelPos,
                    I_InLock_MyBool := #I_InLock_MyBool,
                    I_HMI_bEnableAxis := #IF_HMI.I_Control.I_HMI_bEnableAxis,
                    I_HMI_bResetAxis := #IF_HMI.I_Control.I_HMI_bResetAxis,
                    I_HMI_bjogForward := #IF_HMI.I_Control.I_HMI_bjogForward,
                    I_HMI_bjogBackward := #IF_HMI.I_Control.I_HMI_bjogBackward,
                    I_HMI_bmoveVelocity := #IF_HMI.I_Control.I_HMI_bmoveVelocity,
                    I_HMI_bstop := #IF_HMI.I_Control.I_HMI_bstop,
                    I_HMI_bfastStop := #IF_HMI.I_Control.I_HMI_bfastStop,
                    I_HMI_bHoming := #IF_HMI.I_Control.I_HMI_bHoming,
                    I_HMI_bGoToPos := #IF_HMI.I_Control.I_HMI_bGoToPos,
                    I_HMI_iGoToPos := #IF_HMI.I_Control.I_HMI_iGoToPos,
                    I_HMI_bCallAbsPos := #IF_HMI.I_Control.I_HMI_bCallAbsPos,
                    I_HMI_bRelPos := #IF_HMI.I_Control.I_HMI_bRelPos,
                    I_HMI_MyBool := #IF_HMI.I_Control.I_HMI_MyBool,
                    I_CMD_bGoToPos_0 := #I_CMD_bGoToPos_0,
                    I_InLock_bGoToPos_0 := #I_InLock_bGoToPos_0,
                    I_HMI_bGoToPos_0 := #IF_HMI.I_Control.I_HMI_bGoToPos_0,
                    I_CMD_bGoToPos_1 := #I_CMD_bGoToPos_1,
                    I_InLock_bGoToPos_1 := #I_InLock_bGoToPos_1,
                    I_HMI_bGoToPos_1 := #IF_HMI.I_Control.I_HMI_bGoToPos_1,
                    I_CMD_bGoToPos_2 := #I_CMD_bGoToPos_2,
                    I_InLock_bGoToPos_2 := #I_InLock_bGoToPos_2,
                    I_HMI_bGoToPos_2 := #IF_HMI.I_Control.I_HMI_bGoToPos_2,
                    I_CMD_bGoToPos_3 := #I_CMD_bGoToPos_3,
                    I_InLock_bGoToPos_3 := #I_InLock_bGoToPos_3,
                    I_HMI_bGoToPos_3 := #IF_HMI.I_Control.I_HMI_bGoToPos_3,
                    I_CMD_bGoToPos_4 := #I_CMD_bGoToPos_4,
                    I_InLock_bGoToPos_4 := #I_InLock_bGoToPos_4,
                    I_HMI_bGoToPos_4 := #IF_HMI.I_Control.I_HMI_bGoToPos_4,
                    I_CMD_bGoToPos_5 := #I_CMD_bGoToPos_5,
                    I_InLock_bGoToPos_5 := #I_InLock_bGoToPos_5,
                    I_HMI_bGoToPos_5 := #IF_HMI.I_Control.I_HMI_bGoToPos_5,
                    I_CMD_bGoToPos_6 := #I_CMD_bGoToPos_6,
                    I_InLock_bGoToPos_6 := #I_InLock_bGoToPos_6,
                    I_HMI_bGoToPos_6 := #IF_HMI.I_Control.I_HMI_bGoToPos_6,
                    I_CMD_bGoToPos_7 := #I_CMD_bGoToPos_7,
                    I_InLock_bGoToPos_7 := #I_InLock_bGoToPos_7,
                    I_HMI_bGoToPos_7 := #IF_HMI.I_Control.I_HMI_bGoToPos_7,
                    I_CMD_bGoToPos_8 := #I_CMD_bGoToPos_8,
                    I_InLock_bGoToPos_8 := #I_InLock_bGoToPos_8,
                    I_HMI_bGoToPos_8 := #IF_HMI.I_Control.I_HMI_bGoToPos_8,
                    I_Para_rJog_Speed := #IF_HMI.Parametet.Para_rJog_Speed,
                    I_Para_rMV_Speed := #IF_HMI.Parametet.Para_rMV_Speed,
                    I_Para_rStop_Dec := #IF_HMI.Parametet.Para_rStop_Dec,
                    I_Para_rEStop_Dec := #IF_HMI.Parametet.Para_rEStop_Dec,
                    I_Para_rPos_Abs := #IF_HMI.Parametet.Para_rPos_Abs,
                    I_Para_rSpeed_Abs := #IF_HMI.Parametet.Para_rSpeed_Abs,
                    I_Para_rAcc_Set := #IF_HMI.Parametet.Para_rAcc_Set,
                    I_Para_rDec_Set := #IF_HMI.Parametet.Para_rDec_Set,
                    I_Para_rJerk_Set := #IF_HMI.Parametet.Para_rJerk_Set,
                    O_Status_bAxisReady => #O_Status_bAxisReady,
                    O_Status_bAxisEnabled => #O_Status_bAxisEnabled,
                    O_Status_bjogForward => #O_Status_bjogForward,
                    O_Status_bjogBackward => #O_Status_bjogBackward,
                    O_Status_bHomed => #HOMIEDONE,
                    O_Status_bAtHome => #O_Status_bAtHome,
                    O_Status_bSstill => #O_Status_bSstill,
                    O_Status_bAxisBusy => #O_Status_bAxisBusy,
                    O_Status_bAxisSyned => #O_Status_bAxisSyned,
                    O_Status_bAxisError => #O_Status_bAxisError,
                    O_Status_bAtPos => #O_Status_bAtPos,
                    O_Status_bPosDone => #O_Status_bPosDone,
                    O_Status_bPosing => #O_Status_bPosing,
                    O_Status_bRelPosDone => #O_Status_bRelPosDone,
                    O_Status_rActPos => #O_Status_rActPos,
                    O_Status_rActSpeed => #O_Status_rActSpeed,
                    O_Status_iAxisFaultNum => #O_Status_iAxisFaultNum,
                    O_Status_iDriveFaultNum => #O_Status_iDriveFaultNum,
                    O_Status_iFBStatus => #O_Status_iFBStatus,
                    O_Status_iMCStatus => #O_Status_iMCStatus,
                    O_Status_rDriveTorque => #O_Status_rDriveTorque,
                    O_Status_rDriveTemp => #O_Status_rDriveTemp,
                    O_Status_rDriveRpm => #O_Status_rDriveRpm,
                    O_Status_AxisName => #O_Status_AxisName,
                    O_Status_mybool => #O_Status_mybool,
                    O_Status_myLreal => #O_Status_myLreal);
END_REGION

REGION Network 2 (SCL)
   IF #HOMIEDONE THEN
       #O_Status_bHomed := 1;
   END_IF;
   IF #O_Status_rActSpeed>0.5 THEN
           #O_Status_bHomed := 0;
   END_IF;
END_REGION

REGION Network 4 (SCL)


       "dGlobal".gi_Axis_AbsNum[#Axis_Nr] := #Axis_AbsNum;
END_REGION

REGION Network 6 (SCL)

       "dStruct_Axis".gs_Axis[#Axis_Nr].I_CMD.bResetAxis := #Opmode.Reset;
       "dStruct_Axis".gs_Axis[#Axis_Nr].I_InLock.bjogForward := "dStruct_Axis".gs_Axis[#Axis_Nr].O_Status.bAxisEnabled;
       "dStruct_Axis".gs_Axis[#Axis_Nr].I_InLock.bjogBackward := "dStruct_Axis".gs_Axis[#Axis_Nr].O_Status.bAxisEnabled;
       "dStruct_Axis".gs_Axis[#Axis_Nr].I_InLock.bHoming := true;
       FOR #j := 0 TO 16 DO
           "dStruct_Axis".gs_Axis[#Axis_Nr].I_InLock.bGoToPos[#j] := true;
       END_FOR;


       IF "dGlobal".Old_Pos_Select <> "dGlobal".gbo_Pos_Select THEN//刚切换
           "dStruct_Axis".gs_Axis[0].I_Para.rPos_Abs[0] := "dStruct_Axis".gs_Axis["dGlobal".gbo_Axis_Select].I_Para.rPos_Abs["dGlobal".gbo_Pos_Select];
           "dStruct_Axis".gs_Axis[0].I_Para.rSpeed_Abs[0] := "dStruct_Axis".gs_Axis["dGlobal".gbo_Axis_Select].I_Para.rSpeed_Abs["dGlobal".gbo_Pos_Select];

           "dGlobal".Old_Pos_Select := "dGlobal".gbo_Pos_Select;
       ELSE
           "dStruct_Axis".gs_Axis["dGlobal".gbo_Axis_Select].I_Para.rPos_Abs["dGlobal".gbo_Pos_Select] := "dStruct_Axis".gs_Axis[0].I_Para.rPos_Abs[0];
           "dStruct_Axis".gs_Axis["dGlobal".gbo_Axis_Select].I_Para.rSpeed_Abs["dGlobal".gbo_Pos_Select] := "dStruct_Axis".gs_Axis[0].I_Para.rSpeed_Abs[0];
       END_IF;
END_REGION

REGION Network 7 (SCL)
   #IF_HMI.Show_Sensor.I_SS_bHome := #I_SS_bHome;
   #IF_HMI.Show_Sensor.I_SS_bFW := #I_SS_bFW;
   #IF_HMI.Show_Sensor.I_SS_bBW := #I_SS_bBW;
   #IF_HMI.O_Status.O_Status_bAxisReady := #O_Status_bAxisReady;
   #IF_HMI.O_Status.O_Status_bAxisEnabled := #O_Status_bAxisEnabled;
   #IF_HMI.O_Status.O_Status_bjogForward := #O_Status_bjogForward;
   #IF_HMI.O_Status.O_Status_bjogBackward := #O_Status_bjogBackward;
   #IF_HMI.O_Status.O_Status_bHomed := #O_Status_bHomed;
   #IF_HMI.O_Status.O_Status_bAtHome := #O_Status_bAtHome;
   #IF_HMI.O_Status.O_Status_bSstill := #O_Status_bSstill;
   #IF_HMI.O_Status.O_Status_bAxisBusy := #O_Status_bAxisBusy;
   #IF_HMI.O_Status.O_Status_bAxisSyned := #O_Status_bAxisSyned;
   #IF_HMI.O_Status.O_Status_bAxisError := #O_Status_bAxisError;
   #IF_HMI.O_Status.O_Status_bAtPos := #O_Status_bAtPos;
   #IF_HMI.O_Status.O_Status_bPosDone := #O_Status_bPosDone;
   #IF_HMI.O_Status.O_Status_bPosing := #O_Status_bPosing;
   #IF_HMI.O_Status.O_Status_bRelPosDone := #O_Status_bRelPosDone;
   #IF_HMI.O_Status.O_Status_rActPos := #O_Status_rActPos;
   #IF_HMI.O_Status.O_Status_rActSpeed := #O_Status_rActSpeed;
   #IF_HMI.O_Status.O_Status_iAxisFaultNum := #O_Status_iAxisFaultNum;
   #IF_HMI.O_Status.O_Status_iDriveFaultNum := #O_Status_iDriveFaultNum;
   #IF_HMI.O_Status.O_Status_iFBStatus := #O_Status_iFBStatus;
   #IF_HMI.O_Status.O_Status_iMCStatus := #O_Status_iMCStatus;
   #IF_HMI.O_Status.O_Status_rDriveTorque := #O_Status_rDriveTorque;
   #IF_HMI.O_Status.O_Status_rDriveTemp := #O_Status_rDriveTemp;
   #IF_HMI.O_Status.O_Status_rDriveRpm := #O_Status_rDriveRpm;
   #IF_HMI.O_Status.O_Status_AxisName := #O_Status_AxisName;
   #IF_HMI.O_Status.O_Status_mybool := #O_Status_mybool;
   #IF_HMI.O_Status.O_Status_myLreal := #O_Status_myLreal;
   #IF_HMI.Plant_Identifier := #Plant_Identifier;
END_REGION

REGION Network 8 (SCL)
   "dGlobal".gi_Axis_AbsNum[0] := "dGlobal".gi_Axis_AbsNum["dGlobal".gbo_Axis_Select];
END_REGION
END_FUNCTION_BLOCK

FUNCTION_BLOCK "FB_Pos16_IO"   // FB30142, LAD
{ S7_Optimized_Access := 'TRUE' }
// stored: AutoNumber false, MemoryReserve 100, SetENOAutomatically false
   VAR_INPUT
      Opmode { ExternalAccessible := 'False'; ExternalVisible := 'False'; ExternalWritable := 'False'} : "OPMODE_OUT_UDT";
      TO_PosAxis : TO_PositioningAxis;
      I_iNum_Abspos : Int;
      I_bMan_Enable : Bool;
      I_SS_bHome : Bool;   // 原点传感器
      I_SS_bFW : Bool := TRUE;   // 前限位
      I_SS_bBW : Bool := TRUE;   // 后限位
      I_CMD_bEnableAxis : Bool;   // 使能
      I_CMD_bResetAxis : Bool;   // 复位
      I_CMD_bjogForward : Bool;   // Taster Aufwärts / 正点
      I_CMD_bjogBackward : Bool;   // Taster Abwärts / 反点
      I_CMD_bmoveVelocity : Bool;   // 速度运行
      I_CMD_bstop : Bool;   // 停止
      I_CMD_bfastStop : Bool;   // 急停
      I_CMD_bHoming : Bool;   // 回零
      I_CMD_bGoToPos : Array[0..15] of Bool;   // Start Aufwärts in Automatik / 16个定位
      I_CMD_iGoToPos : Word;   // 16个定位 Word
      I_CMD_bCallAbsPos : Bool;   // 定位位置切换时，单独的定位按钮
      I_CMD_bRelPos : Bool;   // 相对定位
      I_InLock_bEnableAxis : Bool;   // 使能
      I_InLock_bResetAxis : Bool;   // 复位
      I_InLock_bjogForward : Bool;   // Taster Aufwärts / 正点
      I_InLock_bjogBackward : Bool;   // Taster Abwärts / 反点
      I_InLock_bmoveVelocity : Bool;   // 速度运行
      I_InLock_bstop : Bool;   // 停止
      I_InLock_bfastStop : Bool;   // 急停
      I_InLock_bHoming : Bool;   // 回零
      I_InLock_bGoToPos : Array[0..16] of Bool;   // Start Aufwärts in Automatik / 16个定位
      I_InLock_iGoToPos : Word;   // 16个定位 Word
      I_InLock_bCallAbsPos : Bool;   // 定位位置切换时，单独的定位按钮
      I_InLock_bRelPos : Bool;   // 相对定位
      I_InLock_MyBool : Array[0..5] of Bool;   // 临时变量
      I_HMI_bEnableAxis : Bool;   // 使能
      I_HMI_bResetAxis : Bool;   // 复位
      I_HMI_bjogForward : Bool;   // Taster Aufwärts / 正点
      I_HMI_bjogBackward : Bool;   // Taster Abwärts / 反点
      I_HMI_bmoveVelocity : Bool;   // 速度运行
      I_HMI_bstop : Bool;   // 停止
      I_HMI_bfastStop : Bool;   // 急停
      I_HMI_bHoming : Bool;   // 回零
      I_HMI_bGoToPos : Array[0..16] of Bool;   // Start Aufwärts in Automatik / 16个定位
      I_HMI_iGoToPos : Word;   // 16个定位 Word
      I_HMI_bCallAbsPos : Bool;   // 定位位置切换时，单独的定位按钮
      I_HMI_bRelPos : Bool;   // 相对定位
      I_HMI_MyBool : Array[0..5] of Bool;   // 临时变量
      I_CMD_bGoToPos_0 : Bool;   // Start Aufwärts in Automatik / 16个定位自动
      I_InLock_bGoToPos_0 : Bool;   // Start Aufwärts in Automatik / 16个定位条件
      I_HMI_bGoToPos_0 : Bool;   // Start Aufwärts in Automatik / 16个定位HMI
      I_CMD_bGoToPos_1 : Bool;   // Start Aufwärts in Automatik / 16个定位自动
      I_InLock_bGoToPos_1 : Bool;   // Start Aufwärts in Automatik / 16个定位条件
      I_HMI_bGoToPos_1 : Bool;   // Start Aufwärts in Automatik / 16个定位HMI
      I_CMD_bGoToPos_2 : Bool;   // Start Aufwärts in Automatik / 16个定位自动
      I_InLock_bGoToPos_2 : Bool;   // Start Aufwärts in Automatik / 16个定位条件
      I_HMI_bGoToPos_2 : Bool;   // Start Aufwärts in Automatik / 16个定位HMI
      I_CMD_bGoToPos_3 : Bool;   // Start Aufwärts in Automatik / 16个定位自动
      I_InLock_bGoToPos_3 : Bool;   // Start Aufwärts in Automatik / 16个定位条件
      I_HMI_bGoToPos_3 : Bool;   // Start Aufwärts in Automatik / 16个定位HMI
      I_CMD_bGoToPos_4 : Bool;   // Start Aufwärts in Automatik / 16个定位自动
      I_InLock_bGoToPos_4 : Bool;   // Start Aufwärts in Automatik / 16个定位条件
      I_HMI_bGoToPos_4 : Bool;   // Start Aufwärts in Automatik / 16个定位HMI
      I_CMD_bGoToPos_5 : Bool;   // Start Aufwärts in Automatik / 16个定位自动
      I_InLock_bGoToPos_5 : Bool;   // Start Aufwärts in Automatik / 16个定位条件
      I_HMI_bGoToPos_5 : Bool;   // Start Aufwärts in Automatik / 16个定位HMI
      I_CMD_bGoToPos_6 : Bool;   // Start Aufwärts in Automatik / 16个定位自动
      I_InLock_bGoToPos_6 : Bool;   // Start Aufwärts in Automatik / 16个定位条件
      I_HMI_bGoToPos_6 : Bool;   // Start Aufwärts in Automatik / 16个定位HMI
      I_CMD_bGoToPos_7 : Bool;   // Start Aufwärts in Automatik / 16个定位自动
      I_InLock_bGoToPos_7 : Bool;   // Start Aufwärts in Automatik / 16个定位条件
      I_HMI_bGoToPos_7 : Bool;   // Start Aufwärts in Automatik / 16个定位HMI
      I_CMD_bGoToPos_8 : Bool;   // Start Aufwärts in Automatik / 16个定位自动
      I_InLock_bGoToPos_8 : Bool;   // Start Aufwärts in Automatik / 16个定位条件
      I_HMI_bGoToPos_8 : Bool;   // Start Aufwärts in Automatik / 16个定位HMI
   END_VAR
   VAR_OUTPUT
      O_Status_bAxisReady : Bool;   // 轴通讯正常
      O_Status_bAxisEnabled : Bool;   // 轴使能
      O_Status_bjogForward : Bool;   // 轴正点中
      O_Status_bjogBackward : Bool;   // 轴反点中
      O_Status_bHomed : Bool;   // 轴归零完成
      O_Status_bAtHome : Bool;   // 轴在零位
      O_Status_bSstill : Bool;   // 轴静止
      O_Status_bAxisBusy : Bool;   // 轴运行中
      O_Status_bAxisSyned : Bool;   // 同步上
      O_Status_bAxisError : Bool;   // 轴报警
      O_Status_bAtPos : Array[0..15] of Bool;   // Ausgang Aufwärts / 在目标位置上
      O_Status_bPosDone : Array[0..15] of Bool;   // 定位完成
      O_Status_bPosing : Array[0..15] of Bool;   // Ausgang Aufwärts / 定位中
      O_Status_bRelPosDone : Bool;   // 相对定位完成
      O_Status_rActPos : LReal;   // 实际位置
      O_Status_rActSpeed : LReal;   // 实际速度
      O_Status_iAxisFaultNum : UDInt;   // 轴报警代码
      O_Status_iDriveFaultNum : UDInt;   // 驱动报警代码
      O_Status_iFBStatus : Word;   // 运动功能块状态
      O_Status_iMCStatus : Word;   // 运动指令状态
      O_Status_rDriveTorque : LReal;   // 驱动扭矩
      O_Status_rDriveTemp : LReal;   // 驱动温度
      O_Status_rDriveRpm : LReal;   // 驱动转速
      O_Status_AxisName : WString[24] := WSTRING#'No axis';   // Name of axis
      O_Status_mybool : Array[0..5] of Bool;   // 备用
      O_Status_myLreal : Array[0..5] of LReal;   // 备用
   END_VAR
   VAR_IN_OUT
      I_Para_rJog_Speed : Array[0..2] of LReal;   // 点动速度/ACC/DEC/JERK
      I_Para_rMV_Speed : Array[0..2] of LReal;   // 速度运行速度/ACC/DEC/JERK
      I_Para_rStop_Dec : Array[0..1] of LReal;   // 速度运行速度/ACC/DEC/JERK
      I_Para_rEStop_Dec : Array[0..1] of LReal;   // 速度运行速度/ACC/DEC/JERK
      I_Para_iNum_Abspos : Int := 4;
      I_Para_rPos_Abs : Array[0..16] of LReal;   // 绝对定位目标位置 / Over travel switch set
      I_Para_rSpeed_Abs : Array[0..16] of LReal;   // Endlage Unten / 绝对定位速度
      I_Para_rAcc_Set : Array[0..16] of LReal;   // 绝对定位加速度 / Overtravel switch Reset
      I_Para_rDec_Set : Array[0..16] of LReal;   // 绝对定位减速度 / Belt check sensor
      I_Para_rJerk_Set : Array[0..16] of LReal;   // 绝对定位加加速度
      I_Para_rSpeedPercent : LReal := 20.0;   // Endlage Unten / 速度设定百分比
   END_VAR
   VAR
      instAxis01 { ExternalAccessible := 'False'; ExternalVisible := 'False'; ExternalWritable := 'False'} : "LAxisCtrl_PosAxis";
      instShearAxisStatus { S7_SetPoint := 'True'} : "LAxisCtrl_GetAxisStatusWord";
      RT_Reset { S7_SetPoint := 'True'} : R_TRIG;
      RT_PB { ExternalAccessible := 'False'; ExternalVisible := 'False'; ExternalWritable := 'False'} : Array[0..19] of R_TRIG;   // Störungen / Alarms
      FT_PB { ExternalAccessible := 'False'; ExternalVisible := 'False'; ExternalWritable := 'False'; S7_SetPoint := 'True'} : Array[0..19] of F_TRIG;   // Störungen unterdrücken, Belegung identisch mit "Alarm" / Hide Alarms, identical with "Alarm"
      TON_PB { ExternalAccessible := 'False'; ExternalVisible := 'False'; ExternalWritable := 'False'} : Array[0..19] of TON_TIME;   // Fallende Flanke / Falling edge
      TOF_PB { ExternalAccessible := 'False'; ExternalVisible := 'False'; ExternalWritable := 'False'} : Array[0..19] of TOF_TIME;   // Negativer Impuls / Negative pulse
      i { S7_SetPoint := 'True'} : Int;
      temp_cmd_bEnableAxis { ExternalAccessible := 'False'; ExternalVisible := 'False'; ExternalWritable := 'False'} : Bool;
      temp_cmd_bresetAxis { ExternalAccessible := 'False'; ExternalVisible := 'False'; ExternalWritable := 'False'} : Bool;
      temp_cmd_bjogForward { ExternalAccessible := 'False'; ExternalVisible := 'False'; ExternalWritable := 'False'} : Bool;
      temp_cmd_bjogBackward { ExternalAccessible := 'False'; ExternalVisible := 'False'; ExternalWritable := 'False'} : Bool;
      temp_cmd_bmoveVelocity { ExternalAccessible := 'False'; ExternalVisible := 'False'; ExternalWritable := 'False'} : Bool;
      temp_cmd_bstop { ExternalAccessible := 'False'; ExternalVisible := 'False'; ExternalWritable := 'False'} : Bool;
      temp_cmd_bfastStop { ExternalAccessible := 'False'; ExternalVisible := 'False'; ExternalWritable := 'False'} : Bool;
      temp_cmd_bhoming { ExternalAccessible := 'False'; ExternalVisible := 'False'; ExternalWritable := 'False'} : Bool;
      temp_cmd_bGoToPos { ExternalAccessible := 'False'; ExternalVisible := 'False'; ExternalWritable := 'False'} : Array[0..16] of Bool;
      temp_cmd_iGoToPos : Word;
      temp_cmd_bCallAbsPos : Bool;
      temp_cmd_bRelPos : Bool;
      temp_Para_rJog_Speed { ExternalAccessible := 'False'; ExternalVisible := 'False'; ExternalWritable := 'False'} : LReal;
      temp_configuration { ExternalAccessible := 'False'; ExternalVisible := 'False'; ExternalWritable := 'False'} : "LAxisCtrl_typeAxisConfig";   // Diagnostics structure
      temp_Status { ExternalAccessible := 'False'; ExternalVisible := 'False'; ExternalWritable := 'False'} : Word;
      temp_AxisEnabled { ExternalAccessible := 'False'; ExternalVisible := 'False'; ExternalWritable := 'False'} : Bool;
      temp_CommandBusy { ExternalAccessible := 'False'; ExternalVisible := 'False'; ExternalWritable := 'False'} : Bool;
      temp_CommandDone { ExternalAccessible := 'False'; ExternalVisible := 'False'; ExternalWritable := 'False'} : Bool;
      temp_CommandAborted { ExternalAccessible := 'False'; ExternalVisible := 'False'; ExternalWritable := 'False'} : Bool;
      temp_InVelocity { ExternalAccessible := 'False'; ExternalVisible := 'False'; ExternalWritable := 'False'} : Bool;
      temp_jogSelected { ExternalAccessible := 'False'; ExternalVisible := 'False'; ExternalWritable := 'False'} : Bool;
      tempPosAbsoluteSelected { ExternalAccessible := 'False'; ExternalVisible := 'False'; ExternalWritable := 'False'} : Bool;
      temp_diagnostics { ExternalAccessible := 'False'; ExternalVisible := 'False'; ExternalWritable := 'False'} : "LAxisCtrl_typeDiagnostics";
      temp_stop_Dec { ExternalAccessible := 'False'; ExternalVisible := 'False'; ExternalWritable := 'False'} : LReal;
      temp_faststop_Dec { ExternalAccessible := 'False'; ExternalVisible := 'False'; ExternalWritable := 'False'} : LReal;
      temp_cmd_bGoToPosAll : Bool;
      temp_iFBStatus : Word;
      temp_iMCStatus : Word;
      old_iFBStatus : Word;
      old_iMCStatus : Word;
   END_VAR
BEGIN

REGION Network 1
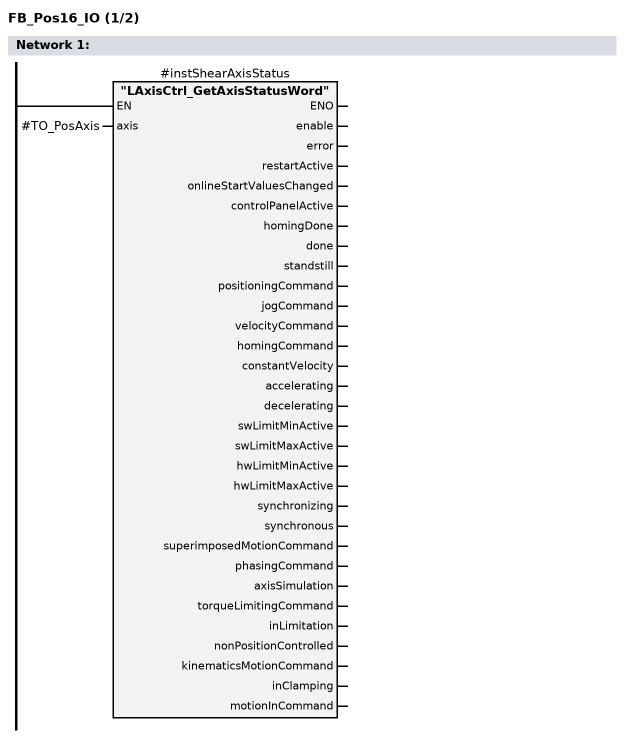
   RUNG wire#powerrail
      #instShearAxisStatus(axis := #TO_PosAxis, enable =>, error =>, restartActive =>, onlineStartValuesChanged =>, controlPanelActive =>, homingDone =>, done =>, standstill =>, positioningCommand =>, jogCommand =>, velocityCommand =>, homingCommand =>, constantVelocity =>, accelerating =>, decelerating =>, swLimitMinActive =>, swLimitMaxActive =>, hwLimitMinActive =>, hwLimitMaxActive =>, synchronizing =>, synchronous =>, superimposedMotionCommand =>, phasingCommand =>, axisSimulation =>, torqueLimitingCommand =>, inLimitation =>, nonPositionControlled =>, kinematicsMotionCommand =>, inClamping =>, motionInCommand =>)
   END_RUNG
   // the same network as SCL:
   #instShearAxisStatus(axis := #TO_PosAxis);   // "LAxisCtrl_GetAxisStatusWord"
END_REGION

REGION Network 2: LAxisCtrl
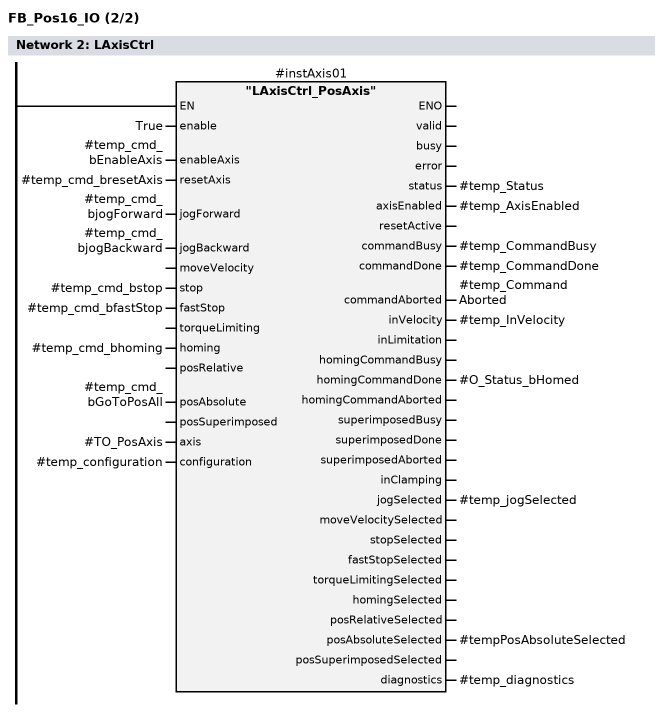
   RUNG wire#powerrail
      #instAxis01(enable := True, enableAxis := #temp_cmd_bEnableAxis, resetAxis := #temp_cmd_bresetAxis, jogForward := #temp_cmd_bjogForward, jogBackward := #temp_cmd_bjogBackward, moveVelocity :=, stop := #temp_cmd_bstop, fastStop := #temp_cmd_bfastStop, torqueLimiting :=, homing := #temp_cmd_bhoming, posRelative :=, posAbsolute := #temp_cmd_bGoToPosAll, posSuperimposed :=, axis := #TO_PosAxis, configuration := #temp_configuration, valid =>, busy =>, error =>, status => #temp_Status, axisEnabled => #temp_AxisEnabled, resetActive =>, commandBusy => #temp_CommandBusy, commandDone => #temp_CommandDone, commandAborted => #temp_CommandAborted, inVelocity => #temp_InVelocity, inLimitation =>, homingCommandBusy =>, homingCommandDone => #O_Status_bHomed, homingCommandAborted =>, superimposedBusy =>, superimposedDone =>, superimposedAborted =>, inClamping =>, jogSelected => #temp_jogSelected, moveVelocitySelected =>, stopSelected =>, fastStopSelected =>, torqueLimitingSelected =>, homingSelected =>, posRelativeSelected =>, posAbsoluteSelected => #tempPosAbsoluteSelected, posSuperimposedSelected =>, diagnostics => #temp_diagnostics)
   END_RUNG
   // the same network as SCL:
   #instAxis01(enable := True,   // "LAxisCtrl_PosAxis"
               enableAxis := #temp_cmd_bEnableAxis,
               resetAxis := #temp_cmd_bresetAxis,
               jogForward := #temp_cmd_bjogForward,
               jogBackward := #temp_cmd_bjogBackward,
               stop := #temp_cmd_bstop,
               fastStop := #temp_cmd_bfastStop,
               homing := #temp_cmd_bhoming,
               posAbsolute := #temp_cmd_bGoToPosAll,
               axis := #TO_PosAxis,
               configuration := #temp_configuration,
               status => #temp_Status,
               axisEnabled => #temp_AxisEnabled,
               commandBusy => #temp_CommandBusy,
               commandDone => #temp_CommandDone,
               commandAborted => #temp_CommandAborted,
               inVelocity => #temp_InVelocity,
               homingCommandDone => #O_Status_bHomed,
               jogSelected => #temp_jogSelected,
               posAbsoluteSelected => #tempPosAbsoluteSelected,
               diagnostics => #temp_diagnostics);
END_REGION

REGION Network 3 (SCL): input
   #temp_cmd_bEnableAxis  := #I_CMD_bEnableAxis OR (#I_HMI_bEnableAxis AND #I_bMan_Enable);
   #temp_cmd_bresetAxis   := #I_CMD_bResetAxis;
   #temp_cmd_bjogForward  := #I_InLock_bjogForward AND (#I_CMD_bjogForward OR (#I_HMI_bjogForward AND #I_bMan_Enable));
   #temp_cmd_bjogBackward := #I_InLock_bjogBackward AND (#I_CMD_bjogBackward OR (#I_HMI_bjogBackward AND #I_bMan_Enable));
   #temp_cmd_bstop        := #I_CMD_bstop OR (#I_HMI_bstop AND #I_bMan_Enable);
   #temp_cmd_bfastStop    := #I_CMD_bfastStop;
   #temp_cmd_bhoming      := #I_InLock_bHoming AND (#I_CMD_bHoming OR #I_HMI_bHoming);
END_REGION

REGION Network 4 (SCL): Configuration
   //#I_Para_rJog_Speed[0] := 10.0;
   #I_Para_rMV_Speed[0]  := 10.0;
   #I_Para_rStop_Dec[0]  := 20.0;
   #I_Para_rEStop_Dec[0] := 50.0;

   #I_Para_rJog_Speed[1] := 10.0 * #I_Para_rJog_Speed[0];
   #I_Para_rJog_Speed[2] := 10.0 * #I_Para_rJog_Speed[0];
   #I_Para_rMV_Speed[1] := 10.0 * #I_Para_rMV_Speed[0];
   #I_Para_rMV_Speed[2] := 10.0 * #I_Para_rMV_Speed[0];
   #I_Para_rStop_Dec[1] := 100.0 * #I_Para_rStop_Dec[0];
   #I_Para_rEStop_Dec[1] := 100.0 * #I_Para_rEStop_Dec[0];

   IF #temp_configuration.jog.velocity <> #I_Para_rJog_Speed[0] OR
       #temp_configuration.jog.acceleration <> #I_Para_rJog_Speed[1] OR
       #temp_configuration.jog.deceleration <> #I_Para_rJog_Speed[2] OR
       #temp_configuration.moveVelocity.acceleration <> #I_Para_rMV_Speed[0] OR
       #temp_configuration.moveVelocity.deceleration <> #I_Para_rMV_Speed[1] OR
       #temp_configuration.moveVelocity.acceleration <> #I_Para_rMV_Speed[2] OR
       #temp_configuration.stop.deceleration <> #I_Para_rStop_Dec[0] OR
       #temp_configuration.stop.jerk <> #I_Para_rStop_Dec[1] OR
       #temp_configuration.fastStop.deceleration <> #I_Para_rEStop_Dec[0] OR
       #temp_configuration.fastStop.jerk <> #I_Para_rEStop_Dec[1]
   THEN
       // Jog
       #temp_configuration.jog.velocity := #I_Para_rJog_Speed[0];
       #temp_configuration.jog.acceleration := #I_Para_rJog_Speed[1];
       #temp_configuration.jog.deceleration := #I_Para_rJog_Speed[2];
       // Move
       #temp_configuration.moveVelocity.velocity := #I_Para_rMV_Speed[0];
       #temp_configuration.moveVelocity.acceleration := #I_Para_rMV_Speed[1];
       #temp_configuration.moveVelocity.deceleration := #I_Para_rMV_Speed[2];
       // Stop   
       #temp_configuration.stop.deceleration := #I_Para_rStop_Dec[0];
       #temp_configuration.stop.jerk := #I_Para_rStop_Dec[1];
       //faststoo
       #temp_configuration.fastStop.deceleration := #I_Para_rEStop_Dec[0];
       #temp_configuration.fastStop.jerk := #I_Para_rEStop_Dec[1];
   END_IF;

   // Homing
   #temp_configuration.homing.mode := 3;//I_iHomeMode
   #temp_configuration.homing.position := 0;//I_iHomePos

   //abspos
   FOR #i := 1 TO 16 DO
       #I_Para_rAcc_Set[#i] := 10.0 * #I_Para_rSpeed_Abs[0];
       #I_Para_rDec_Set[#i] := 10.0 * #I_Para_rSpeed_Abs[0];
       #I_Para_rJerk_Set[#i] := 100.0 * #I_Para_rSpeed_Abs[0];
   END_FOR;


   //#temp_posAbsolute := (I_CMD_iGoToPos <> 16#0);
   #temp_cmd_bGoToPos[1] := (((#Opmode.Automatic_active=1 OR #Opmode.SingleStep_active=1) AND #I_CMD_iGoToPos = 1) OR (#Opmode.Manual_active AND  #I_HMI_iGoToPos = 1)) AND #I_InLock_bGoToPos[1];
   #temp_cmd_bGoToPos[2] := (((#Opmode.Automatic_active=1 OR #Opmode.SingleStep_active=1) AND #I_CMD_iGoToPos = 2) OR (#Opmode.Manual_active AND  #I_HMI_iGoToPos = 2)) AND #I_InLock_bGoToPos[2];
   #temp_cmd_bGoToPos[3] := (((#Opmode.Automatic_active=1 OR #Opmode.SingleStep_active=1) AND #I_CMD_iGoToPos = 3) OR (#Opmode.Manual_active AND  #I_HMI_iGoToPos = 3)) AND #I_InLock_bGoToPos[3];
   #temp_cmd_bGoToPos[4] := (((#Opmode.Automatic_active=1 OR #Opmode.SingleStep_active=1) AND #I_CMD_iGoToPos = 4) OR (#Opmode.Manual_active AND  #I_HMI_iGoToPos = 4)) AND #I_InLock_bGoToPos[4];
   #temp_cmd_bGoToPos[5] := (((#Opmode.Automatic_active=1 OR #Opmode.SingleStep_active=1) AND #I_CMD_iGoToPos = 5) OR (#Opmode.Manual_active AND  #I_HMI_iGoToPos = 5)) AND #I_InLock_bGoToPos[5];
   #temp_cmd_bGoToPos[6] := (((#Opmode.Automatic_active=1 OR #Opmode.SingleStep_active=1) AND #I_CMD_iGoToPos = 6) OR (#Opmode.Manual_active AND  #I_HMI_iGoToPos = 6)) AND #I_InLock_bGoToPos[6];
   #temp_cmd_bGoToPos[7] := (((#Opmode.Automatic_active=1 OR #Opmode.SingleStep_active=1) AND #I_CMD_iGoToPos = 7) OR (#Opmode.Manual_active AND  #I_HMI_iGoToPos = 7)) AND #I_InLock_bGoToPos[7];
   #temp_cmd_bGoToPos[8] := (((#Opmode.Automatic_active=1 OR #Opmode.SingleStep_active=1) AND #I_CMD_iGoToPos = 8) OR (#Opmode.Manual_active AND  #I_HMI_iGoToPos = 8)) AND #I_InLock_bGoToPos[8];
   #temp_cmd_bGoToPos[9] := (((#Opmode.Automatic_active=1 OR #Opmode.SingleStep_active=1) AND #I_CMD_iGoToPos = 9) OR (#Opmode.Manual_active AND  #I_HMI_iGoToPos = 9)) AND #I_InLock_bGoToPos[9];
   #temp_cmd_bGoToPos[10] := (((#Opmode.Automatic_active=1 OR #Opmode.SingleStep_active=1) AND #I_CMD_iGoToPos = 10) OR (#Opmode.Manual_active AND  #I_HMI_iGoToPos = 10)) AND #I_InLock_bGoToPos[10];
   #temp_cmd_bGoToPos[11] := (((#Opmode.Automatic_active=1 OR #Opmode.SingleStep_active=1) AND #I_CMD_iGoToPos = 11) OR (#Opmode.Manual_active AND  #I_HMI_iGoToPos = 11)) AND #I_InLock_bGoToPos[11];
   #temp_cmd_bGoToPos[12] := (((#Opmode.Automatic_active=1 OR #Opmode.SingleStep_active=1) AND #I_CMD_iGoToPos = 12) OR (#Opmode.Manual_active AND  #I_HMI_iGoToPos = 12)) AND #I_InLock_bGoToPos[12];
   #temp_cmd_bGoToPos[13] := (((#Opmode.Automatic_active=1 OR #Opmode.SingleStep_active=1) AND #I_CMD_iGoToPos = 13) OR (#Opmode.Manual_active AND  #I_HMI_iGoToPos = 13)) AND #I_InLock_bGoToPos[13];
   #temp_cmd_bGoToPos[14] := (((#Opmode.Automatic_active=1 OR #Opmode.SingleStep_active=1) AND #I_CMD_iGoToPos = 14) OR (#Opmode.Manual_active AND  #I_HMI_iGoToPos = 14)) AND #I_InLock_bGoToPos[14];
   #temp_cmd_bGoToPos[15] := (((#Opmode.Automatic_active=1 OR #Opmode.SingleStep_active=1) AND #I_CMD_iGoToPos = 15) OR (#Opmode.Manual_active AND  #I_HMI_iGoToPos = 15)) AND #I_InLock_bGoToPos[15];
   #temp_cmd_bGoToPos[16] := (((#Opmode.Automatic_active=1 OR #Opmode.SingleStep_active=1) AND #I_CMD_iGoToPos = 16) OR (#Opmode.Manual_active AND  #I_HMI_iGoToPos = 16)) AND #I_InLock_bGoToPos[16];

   #temp_cmd_bGoToPosAll := #temp_cmd_bGoToPos[1] OR #temp_cmd_bGoToPos[2] OR #temp_cmd_bGoToPos[3] OR #temp_cmd_bGoToPos[4]
   OR #temp_cmd_bGoToPos[5] OR #temp_cmd_bGoToPos[6] OR #temp_cmd_bGoToPos[7] OR #temp_cmd_bGoToPos[8]
   OR #temp_cmd_bGoToPos[9] OR #temp_cmd_bGoToPos[10] OR #temp_cmd_bGoToPos[11] OR #temp_cmd_bGoToPos[12]
   OR #temp_cmd_bGoToPos[13] OR #temp_cmd_bGoToPos[14] OR #temp_cmd_bGoToPos[15] OR #temp_cmd_bGoToPos[16]
   ;
   //#temp_posAbsolute :=
   //I_bGoToPos[0] OR I_bGoToPos[1] OR I_bGoToPos[2] OR I_bGoToPos[3] OR
   //I_bGoToPos[4] OR I_bGoToPos[5] OR I_bGoToPos[6] OR I_bGoToPos[7] OR
   //I_bGoToPos[8] OR I_bGoToPos[9] OR I_bGoToPos[10] OR I_bGoToPos[11] OR
   //I_bGoToPos[12] OR I_bGoToPos[13] OR I_bGoToPos[14] OR I_bGoToPos[15];

   FOR #i := 1 TO 16 DO
   //    #RT_PB[#i](CLK := I_bGoToPos[#i]);
       #RT_PB[#i](CLK := #temp_cmd_bGoToPos[#i]);

       IF #RT_PB[#i].Q THEN
           #temp_configuration.posAbsolute.position := #I_Para_rPos_Abs[#i];
           #temp_configuration.posAbsolute.velocity := #I_Para_rSpeed_Abs[#i];
           #temp_configuration.posAbsolute.direction := 3;//temp_posAbsolute_direction

           #temp_configuration.posAbsolute.acceleration := #I_Para_rAcc_Set[#i];
           #temp_configuration.posAbsolute.deceleration := #I_Para_rDec_Set[#i];
           #temp_configuration.posAbsolute.jerk := #I_Para_rJerk_Set[#i];

       END_IF;
   END_FOR;
END_REGION

REGION Network 5 (SCL): output
   #O_Status_bAxisReady := true;//#TO_PosAxis.StatusWord.%X1;
   #O_Status_bAxisEnabled := #temp_AxisEnabled;
   #O_Status_bjogForward := #temp_cmd_bjogForward;// AND #temp_jogSelected;
   #O_Status_bjogBackward := #temp_cmd_bjogBackward;// AND #temp_jogSelected;
   //#O_Status_bHomed := #TO_PosAxis.StatusWord.%X5;
   #O_Status_bAxisError := #TO_PosAxis.StatusWord.%X1;
   #O_Status_rActPos := #TO_PosAxis.ActualPosition;
   #O_Status_rActSpeed := #TO_PosAxis.ActualVelocity;
   #O_Status_iAxisFaultNum := #TO_PosAxis.ErrorDetail.Number;
   //O_DriveFaultNum
   //O_Status_iFBStatus := #temp_diagnostics.status;
   //O_Status_iMCStatus := #temp_diagnostics.subfunctionStatus;
   //O_Torque
   //oAxisName  := 

   FOR #i := 0 TO 15 DO
       #O_Status_bAtPos[#i] := "FC_bNearIn"(rAct := #O_Status_rActPos, rTgt := #I_Para_rPos_Abs[#i], rDelta := 1.0, bModule := 0, rModulo := 0);
   END_FOR;

   //O_bPosDone
   //O_bPosing
   //#tempPosAbsoluteSelected
END_REGION

REGION Network 6 (SCL): Reset
   #RT_Reset(CLK := #temp_cmd_bresetAxis);
   IF #RT_Reset.Q THEN
       #O_Status_iFBStatus := 16#00;
       #O_Status_iMCStatus := 16#00;
   END_IF;

   #temp_iFBStatus := #temp_diagnostics.status;
   IF #temp_iFBStatus <> #old_iFBStatus THEN
       #O_Status_iFBStatus := #temp_diagnostics.status;
       #old_iFBStatus := #temp_iFBStatus;
   END_IF;
   #temp_iMCStatus := #temp_diagnostics.subfunctionStatus;
   IF #temp_iMCStatus <> #old_iMCStatus THEN
       #O_Status_iFBStatus := #temp_diagnostics.subfunctionStatus;
       #old_iMCStatus := #temp_iMCStatus;
   END_IF;
END_REGION

REGION Network 7 (SCL)
   (*
   FOR #i := 9 TO 16 DO
       IF #I_iNum_Abspos < #i THEN
           I_InLock_bGoToPos[#i] := false;
       END_IF;
   END_FOR;
   *)
END_REGION
END_FUNCTION_BLOCK

FUNCTION_BLOCK "LAxisCtrl_GetAxisStatusWord"
{ S7_Optimized_Access := 'TRUE' }
AUTHOR : 'tech.team.motioncontrol@siemens.com'
FAMILY : AxisCtrl
VERSION : 1.0
   VAR_INPUT 
      axis {InstructionName := 'TO_SpeedAxis'; LibVersion := '6.0'} : TO_SpeedAxis;
   END_VAR

   VAR_OUTPUT 
      enable { ExternalWritable := 'False'; S7_HiddenAssignment := 'HideIfNoParamAssigned'} : Bool;
      error { ExternalWritable := 'False'; S7_HiddenAssignment := 'HideIfNoParamAssigned'} : Bool;
      restartActive { ExternalWritable := 'False'; S7_HiddenAssignment := 'HideIfNoParamAssigned'} : Bool;
      onlineStartValuesChanged { ExternalWritable := 'False'; S7_HiddenAssignment := 'HideIfNoParamAssigned'} : Bool;
      controlPanelActive { ExternalWritable := 'False'; S7_HiddenAssignment := 'HideIfNoParamAssigned'} : Bool;
      homingDone { ExternalWritable := 'False'; S7_HiddenAssignment := 'HideIfNoParamAssigned'} : Bool;
      done { ExternalWritable := 'False'; S7_HiddenAssignment := 'HideIfNoParamAssigned'} : Bool;
      standstill { ExternalWritable := 'False'; S7_HiddenAssignment := 'HideIfNoParamAssigned'} : Bool;
      positioningCommand { ExternalWritable := 'False'; S7_HiddenAssignment := 'HideIfNoParamAssigned'} : Bool;
      jogCommand { ExternalWritable := 'False'; S7_HiddenAssignment := 'HideIfNoParamAssigned'} : Bool;
      velocityCommand { ExternalWritable := 'False'; S7_HiddenAssignment := 'HideIfNoParamAssigned'} : Bool;
      homingCommand { ExternalWritable := 'False'; S7_HiddenAssignment := 'HideIfNoParamAssigned'} : Bool;
      constantVelocity { ExternalWritable := 'False'; S7_HiddenAssignment := 'HideIfNoParamAssigned'} : Bool;
      accelerating { ExternalWritable := 'False'; S7_HiddenAssignment := 'HideIfNoParamAssigned'} : Bool;
      decelerating { ExternalWritable := 'False'; S7_HiddenAssignment := 'HideIfNoParamAssigned'} : Bool;
      swLimitMinActive { ExternalWritable := 'False'; S7_HiddenAssignment := 'HideIfNoParamAssigned'} : Bool;
      swLimitMaxActive { ExternalWritable := 'False'; S7_HiddenAssignment := 'HideIfNoParamAssigned'} : Bool;
      hwLimitMinActive { ExternalWritable := 'False'; S7_HiddenAssignment := 'HideIfNoParamAssigned'} : Bool;
      hwLimitMaxActive { ExternalWritable := 'False'; S7_HiddenAssignment := 'HideIfNoParamAssigned'} : Bool;
      synchronizing { ExternalWritable := 'False'; S7_HiddenAssignment := 'HideIfNoParamAssigned'} : Bool;
      synchronous { ExternalWritable := 'False'; S7_HiddenAssignment := 'HideIfNoParamAssigned'} : Bool;
      superimposedMotionCommand { ExternalWritable := 'False'; S7_HiddenAssignment := 'HideIfNoParamAssigned'} : Bool;
      phasingCommand { ExternalWritable := 'False'; S7_HiddenAssignment := 'HideIfNoParamAssigned'} : Bool;
      axisSimulation { ExternalWritable := 'False'; S7_HiddenAssignment := 'HideIfNoParamAssigned'} : Bool;
      torqueLimitingCommand { ExternalWritable := 'False'; S7_HiddenAssignment := 'HideIfNoParamAssigned'} : Bool;
      inLimitation { ExternalWritable := 'False'; S7_HiddenAssignment := 'HideIfNoParamAssigned'} : Bool;
      nonPositionControlled { ExternalWritable := 'False'; S7_HiddenAssignment := 'HideIfNoParamAssigned'} : Bool;
      kinematicsMotionCommand { ExternalWritable := 'False'; S7_HiddenAssignment := 'HideIfNoParamAssigned'} : Bool;
      inClamping { ExternalWritable := 'False'; S7_HiddenAssignment := 'HideIfNoParamAssigned'} : Bool;
      motionInCommand { ExternalWritable := 'False'; S7_HiddenAssignment := 'HideIfNoParamAssigned'} : Bool;
   END_VAR

   VAR_TEMP 
      tempStatusWord : DWord;
   END_VAR


BEGIN
	//==========================================================================================
	// SIEMENS AG
	// (c)Copyright 2017 All Rights Reserved
	//------------------------------------------------------------------------------------------
	// Library: LAxisCtrl
	// Tested with: S7-1515T-2 PN
	// Engineering: TIA Portal V15
	// Restrictions: ---
	// Requirements: S7-1500/S7-1500T FW 2.5
	// Functionality: The FB is splitting the status word of an axis into bits.
	// Support: tech.team.motioncontrol@siemens.com
	// Note: Parameter comments are only available in language 'English (United States)'
	//------------------------------------------------------------------------------------------
	// Change log table:
	// Version    Date          Expert in charge    Changes applied
	// 01.00.01   04.10.2016    AL                  First released version
	// 01.00.02   29.03.2017    AL                  Added support information
	// 01.00.04   14.12.2017    RS                  Added new tags of status word
	//===========================================================================================
	
	//----------------------------------------------------------------------------------------------
	// Read statusword
	//----------------------------------------------------------------------------------------------
	#tempStatusWord := #axis.StatusWord;
	
	//----------------------------------------------------------------------------------------------
	// Write outputs
	//----------------------------------------------------------------------------------------------
	#enable := #tempStatusWord.%X0;
	#error := #tempStatusWord.%X1;
	#restartActive := #tempStatusWord.%X2;
	#onlineStartValuesChanged := #tempStatusWord.%X3;
	#controlPanelActive := #tempStatusWord.%X4;
	#homingDone := #tempStatusWord.%X5;
	#done := #tempStatusWord.%X6;
	#standstill := #tempStatusWord.%X7;
	#positioningCommand := #tempStatusWord.%X8;
	#jogCommand := #tempStatusWord.%X9;
	#velocityCommand := #tempStatusWord.%X10;
	#homingCommand := #tempStatusWord.%X11;
	#constantVelocity := #tempStatusWord.%X12;
	#accelerating := #tempStatusWord.%X13;
	#decelerating := #tempStatusWord.%X14;
	#swLimitMinActive := #tempStatusWord.%X15;
	#swLimitMaxActive := #tempStatusWord.%X16;
	#hwLimitMinActive := #tempStatusWord.%X17;
	#hwLimitMaxActive := #tempStatusWord.%X18;
	#synchronizing := #tempStatusWord.%X21;
	#synchronous := #tempStatusWord.%X22;
	#superimposedMotionCommand := #tempStatusWord.%X23;
	#phasingCommand := #tempStatusWord.%X24;
	#axisSimulation := #tempStatusWord.%X25;
	#torqueLimitingCommand := #tempStatusWord.%X26;
	#inLimitation := #tempStatusWord.%X27;
	#nonPositionControlled := #tempStatusWord.%X28;
	#kinematicsMotionCommand := #tempStatusWord.%X29; // V15
	#inClamping := #tempStatusWord.%X30;
	#motionInCommand := #tempStatusWord.%X31; // V15
END_FUNCTION_BLOCK

FUNCTION_BLOCK "LAxisCtrl_PosAxis"
{ S7_Optimized_Access := 'TRUE' }
AUTHOR : 'tech.team.motioncontrol@siemens.com'
FAMILY : AxisCtrl
VERSION : 1.0
   VAR_INPUT 
      enable : Bool := FALSE;
      enableAxis : Bool := FALSE;
      resetAxis : Bool := FALSE;
      jogForward : Bool := FALSE;
      jogBackward : Bool := FALSE;
      moveVelocity : Bool := FALSE;
      stop : Bool := FALSE;
      fastStop : Bool := FALSE;
      torqueLimiting : Bool := FALSE;
      homing : Bool := FALSE;
      posRelative : Bool := FALSE;
      posAbsolute : Bool := FALSE;
      posSuperimposed : Bool := FALSE;
      axis {InstructionName := 'TO_PositioningAxis'; LibVersion := '6.0'} : TO_PositioningAxis;
   END_VAR

